LIN {X 0,Y 523.354,Z 614.089,A -85,B 0,C 180,E1 -4766.919,E2 -4766.919} C_VEL
LIN {X 0,Y 523.269,Z 615.476,A -85,B 0,C 180,E1 -4768.459,E2 -4768.459} C_VEL
LIN {X 0,Y 523.242,Z 616,A -85,B 0,C 180,E1 -4769.998,E2 -4769.998} C_VEL
LIN {X 0,Y 523.268,Z 615.478,A -85,B 0,C 180,E1 -4771.537,E2 -4771.537} C_VEL
LIN {X 0,Y 523.353,Z 614.092,A -85,B 0,C 180,E1 -4773.077,E2 -4773.077} C_VEL
LIN {X 0,Y 523.311,Z 611.636,A -85,B 0,C 180,E1 -4774.62,E2 -4774.62} C_VEL
LIN {X 0,Y 523.409,Z 608.259,A -85,B 0,C 180,E1 -4776.164,E2 -4776.164} C_VEL
LIN {X 0,Y 523.505,Z 602.475,A -85,B 0,C 180,E1 -4778.101,E2 -4778.101} C_VEL
LIN {X 0,Y 523.657,Z 594.794,A -85,B 0,C 180,E1 -4780.046,E2 -4780.046} C_VEL
LIN {X 0,Y 523.952,Z 586.574,A -85,B 0,C 180,E1 -4781.713,E2 -4781.713} C_VEL
LIN {X 0,Y 524.219,Z 576.745,A -85,B 0,C 180,E1 -4783.369,E2 -4783.369} C_VEL
LIN {X 0,Y 524.679,Z 566.039,A -85,B 0,C 180,E1 -4784.883,E2 -4784.883} C_VEL
LIN {X 0,Y 525.131,Z 554.075,A -85,B 0,C 180,E1 -4786.32,E2 -4786.32} C_VEL
LIN {X 0,Y 525.732,Z 541.515,A -85,B 0,C 180,E1 -4787.602,E2 -4787.602} C_VEL
LIN {X 0,Y 526.283,Z 529.069,A -85,B 0,C 180,E1 -4788.69,E2 -4788.69} C_VEL
LIN {X 0,Y 526.86,Z 515.69,A -85,B 0,C 180,E1 -4789.68,E2 -4789.68} C_VEL
LIN {X 0,Y 527.439,Z 501.437,A -85,B 0,C 180,E1 -4790.573,E2 -4790.573} C_VEL
LIN {X 0,Y 528.124,Z 485.316,A -85,B 0,C 180,E1 -4791.395,E2 -4791.395} C_VEL
LIN {X 0,Y 528.599,Z 470.295,A -85,B 0,C 180,E1 -4792.007,E2 -4792.007} C_VEL
LIN {X 0,Y 529.013,Z 454.139,A -85,B 0,C 180,E1 -4792.503,E2 -4792.503} C_VEL
LIN {X 0,Y 529.379,Z 437.934,A -85,B 0,C 180,E1 -4792.847,E2 -4792.847} C_VEL
LIN {X 0,Y 530.879,Z 249.022,A -85,B 0,C 180,E1 -4795.545,E2 -4795.545} C_VEL
LIN {X 0,Y 528.181,Z 233.832,A -85,B 0,C 180,E1 -4795.92,E2 -4795.92} C_VEL
LIN {X 0,Y 529.038,Z 210.019,A -85,B 0,C 180,E1 -4798.165,E2 -4798.165} C_VEL
LIN {X 0,Y 523.914,Z 192.537,A -85,B 0,C 180,E1 -4800.198,E2 -4800.198} C_VEL
LIN {X 0,Y 523.925,Z 192.529,A -85,B 0,C 180,E1 -4803.362,E2 -4803.362} C_VEL
LIN {X 0,Y 523.885,Z 192.538,A -85,B 0,C 180,E1 -4806.399,E2 -4806.399} C_VEL
LIN {X 0,Y 523.902,Z 192.542,A -85,B 0,C 180,E1 -4809.082,E2 -4809.082} C_VEL
LIN {X 0,Y 523.931,Z 192.53,A -85,B 0,C 180,E1 -4812.116,E2 -4812.116} C_VEL
LIN {X 0,Y 523.932,Z 192.533,A -85,B 0,C 180,E1 -4815.307,E2 -4815.307} C_VEL
LIN {X 0,Y 523.947,Z 192.531,A -85,B 0,C 180,E1 -4818.686,E2 -4818.686} C_VEL
LIN {X 0,Y 523.894,Z 192.543,A -85,B 0,C 180,E1 -4821.078,E2 -4821.078} C_VEL
LIN {X 0,Y 523.899,Z 192.532,A -85,B 0,C 180,E1 -4823.826,E2 -4823.826} C_VEL
LIN {X 0,Y 523.914,Z 192.536,A -85,B 0,C 180,E1 -4826.634,E2 -4826.634} C_VEL
LIN {X 0,Y 523.926,Z 192.535,A -85,B 0,C 180,E1 -4829.354,E2 -4829.354} C_VEL
LIN {X 0,Y 523.948,Z 192.528,A -85,B 0,C 180,E1 -4832.279,E2 -4832.279} C_VEL
LIN {X 0,Y 523.922,Z 192.528,A -85,B 0,C 180,E1 -4834.58,E2 -4834.58} C_VEL
LIN {X 0,Y 523.921,Z 192.537,A -85,B 0,C 180,E1 -4837.107,E2 -4837.107} C_VEL
LIN {X 0,Y 523.946,Z 192.52,A -85,B 0,C 180,E1 -4839.865,E2 -4839.865} C_VEL
LIN {X 0,Y 523.937,Z 192.535,A -85,B 0,C 180,E1 -4842.837,E2 -4842.837} C_VEL
LIN {X 0,Y 523.942,Z 192.529,A -85,B 0,C 180,E1 -4845.235,E2 -4845.235} C_VEL
LIN {X 0,Y 523.984,Z 192.514,A -85,B 0,C 180,E1 -4848.394,E2 -4848.394} C_VEL
LIN {X 0,Y 523.973,Z 192.525,A -85,B 0,C 180,E1 -4851.516,E2 -4851.516} C_VEL
LIN {X 0,Y 524.066,Z 192.515,A -85,B 0,C 180,E1 -4854.614,E2 -4854.614} C_VEL
LIN {X 0,Y 524.075,Z 192.505,A -85,B 0,C 180,E1 -4857.695,E2 -4857.695} C_VEL
LIN {X 0,Y 524.096,Z 192.517,A -85,B 0,C 180,E1 -4860.769,E2 -4860.769} C_VEL
LIN {X 0,Y 524.044,Z 192.514,A -85,B 0,C 180,E1 -4863.075,E2 -4863.075} C_VEL
LIN {X 0,Y 524.011,Z 192.518,A -85,B 0,C 180,E1 -4866.16,E2 -4866.16} C_VEL
LIN {X 0,Y 523.972,Z 192.524,A -85,B 0,C 180,E1 -4869.263,E2 -4869.263} C_VEL
LIN {X 0,Y 523.975,Z 192.516,A -85,B 0,C 180,E1 -4871.744,E2 -4871.744} C_VEL
LIN {X 0,Y 523.961,Z 192.527,A -85,B 0,C 180,E1 -4875.054,E2 -4875.054} C_VEL
LIN {X 0,Y 523.935,Z 192.527,A -85,B 0,C 180,E1 -4877.97,E2 -4877.97} C_VEL
LIN {X 0,Y 523.943,Z 192.53,A -85,B 0,C 180,E1 -4880.412,E2 -4880.412} C_VEL
LIN {X 0,Y 523.914,Z 192.534,A -85,B 0,C 180,E1 -4882.894,E2 -4882.894} C_VEL
LIN {X 0,Y 523.955,Z 192.524,A -85,B 0,C 180,E1 -4886.022,E2 -4886.022} C_VEL
LIN {X 0,Y 523.913,Z 192.534,A -85,B 0,C 180,E1 -4888.877,E2 -4888.877} C_VEL
LIN {X 0,Y 523.894,Z 192.532,A -85,B 0,C 180,E1 -4891.546,E2 -4891.546} C_VEL
LIN {X 0,Y 523.915,Z 192.535,A -85,B 0,C 180,E1 -4894.292,E2 -4894.292} C_VEL
LIN {X 0,Y 523.887,Z 192.534,A -85,B 0,C 180,E1 -4897.134,E2 -4897.134} C_VEL
LIN {X 0,Y 523.916,Z 192.532,A -85,B 0,C 180,E1 -4900.132,E2 -4900.132} C_VEL
LIN {X 0,Y 523.917,Z 192.537,A -85,B 0,C 180,E1 -4902.462,E2 -4902.462} C_VEL
LIN {X 0,Y 523.924,Z 192.525,A -85,B 0,C 180,E1 -4905.313,E2 -4905.313} C_VEL
LIN {X 0,Y 523.881,Z 192.536,A -85,B 0,C 180,E1 -4906.946,E2 -4906.946} C_VEL
LIN {X 0,Y 523.223,Z 192.62,A -85,B 0,C 180,E1 -4907.588,E2 -4907.588} C_VEL
LIN {X 0,Y 520.388,Z 192.976,A -85,B 0,C 180,E1 -4908.63,E2 -4908.63} C_VEL
LIN {X 0,Y 517.986,Z 193.277,A -85,B 0,C 180,E1 -4909.47,E2 -4909.47} C_VEL
LIN {X 0,Y 516.951,Z 193.403,A -85,B 0,C 180,E1 -4910.118,E2 -4910.118} C_VEL
LIN {X 0,Y 516.864,Z 193.412,A -85,B 0,C 180,E1 -4910.337,E2 -4910.337} C_VEL
LIN {X 0,Y 516.87,Z 193.41,A -85,B 0,C 180,E1 -4913.345,E2 -4913.345} C_VEL
LIN {X 0,Y 516.897,Z 193.41,A -85,B 0,C 180,E1 -4916.124,E2 -4916.124} C_VEL
LIN {X 0,Y 516.88,Z 193.407,A -85,B 0,C 180,E1 -4918.939,E2 -4918.939} C_VEL
LIN {X 0,Y 516.853,Z 193.413,A -85,B 0,C 180,E1 -4921.584,E2 -4921.584} C_VEL
LIN {X 0,Y 516.867,Z 193.414,A -85,B 0,C 180,E1 -4924.211,E2 -4924.211} C_VEL
LIN {X 0,Y 516.851,Z 193.411,A -85,B 0,C 180,E1 -4926.779,E2 -4926.779} C_VEL
LIN {X 0,Y 516.925,Z 193.409,A -85,B 0,C 180,E1 -4929.738,E2 -4929.738} C_VEL
LIN {X 0,Y 516.876,Z 193.411,A -85,B 0,C 180,E1 -4932.597,E2 -4932.597} C_VEL
LIN {X 0,Y 516.934,Z 193.403,A -85,B 0,C 180,E1 -4935.032,E2 -4935.032} C_VEL
LIN {X 0,Y 516.967,Z 193.402,A -85,B 0,C 180,E1 -4938.236,E2 -4938.236} C_VEL
LIN {X 0,Y 516.931,Z 193.406,A -85,B 0,C 180,E1 -4941.401,E2 -4941.401} C_VEL
LIN {X 0,Y 516.986,Z 193.392,A -85,B 0,C 180,E1 -4944.542,E2 -4944.542} C_VEL
LIN {X 0,Y 517.076,Z 193.391,A -85,B 0,C 180,E1 -4947.665,E2 -4947.665} C_VEL
LIN {X 0,Y 516.9,Z 193.516,A -85,B 0,C 180,E1 -4948.979,E2 -4948.979} C_VEL
LIN {X 0,Y 520.755,Z 207.242,A -85,B 0,C 180,E1 -4950.748,E2 -4950.748} C_VEL
LIN {X 0,Y 522.505,Z 211.957,A -85,B 0,C 180,E1 -4950.917,E2 -4950.917} C_VEL
LIN {X 0,Y 524.594,Z 222.487,A -85,B 0,C 180,E1 -4951.189,E2 -4951.189} C_VEL
LIN {X 0,Y 522.849,Z 412.749,A -85,B 0,C 180,E1 -4953.951,E2 -4953.951} C_VEL
LIN {X 0,Y 522.467,Z 429.792,A -85,B 0,C 180,E1 -4954.356,E2 -4954.356} C_VEL
LIN {X 0,Y 521.978,Z 445.68,A -85,B 0,C 180,E1 -4954.892,E2 -4954.892} C_VEL
LIN {X 0,Y 521.408,Z 461.923,A -85,B 0,C 180,E1 -4955.61,E2 -4955.61} C_VEL
LIN {X 0,Y 520.734,Z 477.792,A -85,B 0,C 180,E1 -4956.492,E2 -4956.492} C_VEL
LIN {X 0,Y 520.007,Z 492.311,A -85,B 0,C 180,E1 -4957.476,E2 -4957.476} C_VEL
LIN {X 0,Y 519.365,Z 505.674,A -85,B 0,C 180,E1 -4958.562,E2 -4958.562} C_VEL
LIN {X 0,Y 518.695,Z 518.158,A -85,B 0,C 180,E1 -4959.753,E2 -4959.753} C_VEL
LIN {X 0,Y 518.085,Z 530.572,A -85,B 0,C 180,E1 -4961.147,E2 -4961.147} C_VEL
LIN {X 0,Y 517.568,Z 541.215,A -85,B 0,C 180,E1 -4962.55,E2 -4962.55} C_VEL
LIN {X 0,Y 517.129,Z 551.521,A -85,B 0,C 180,E1 -4964.161,E2 -4964.161} C_VEL
LIN {X 0,Y 516.818,Z 560.197,A -85,B 0,C 180,E1 -4965.783,E2 -4965.783} C_VEL
LIN {X 0,Y 516.551,Z 567.484,A -85,B 0,C 180,E1 -4967.418,E2 -4967.418} C_VEL
LIN {X 0,Y 516.425,Z 573.496,A -85,B 0,C 180,E1 -4969.065,E2 -4969.065} C_VEL
LIN {X 0,Y 516.314,Z 578.28,A -85,B 0,C 180,E1 -4970.728,E2 -4970.728} C_VEL
LIN {X 0,Y 516.194,Z 581.912,A -85,B 0,C 180,E1 -4972.41,E2 -4972.41} C_VEL
LIN {X 0,Y 516.148,Z 584.516,A -85,B 0,C 180,E1 -4974.175,E2 -4974.175} C_VEL
LIN {X 0,Y 516.147,Z 585.934,A -85,B 0,C 180,E1 -4976.015,E2 -4976.015} C_VEL
LIN {X 0,Y 516.178,Z 586.005,A -85,B 0,C 180,E1 -4977.747,E2 -4977.747} C_VEL
LIN {X 0,Y 516.201,Z 585.047,A -85,B 0,C 180,E1 -4979.383,E2 -4979.383} C_VEL
LIN {X 0,Y 516.198,Z 582.857,A -85,B 0,C 180,E1 -4981.157,E2 -4981.157} C_VEL
LIN {X 0,Y 516.284,Z 579.196,A -85,B 0,C 180,E1 -4982.992,E2 -4982.992} C_VEL
LIN {X 0,Y 516.365,Z 574.005,A -85,B 0,C 180,E1 -4984.866,E2 -4984.866} C_VEL
LIN {X 0,Y 516.566,Z 567.745,A -85,B 0,C 180,E1 -4986.61,E2 -4986.61} C_VEL
LIN {X 0,Y 516.818,Z 560.334,A -85,B 0,C 180,E1 -4988.285,E2 -4988.285} C_VEL
LIN {X 0,Y 517.076,Z 552.855,A -85,B 0,C 180,E1 -4989.704,E2 -4989.704} C_VEL
LIN {X 0,Y 517.478,Z 543.552,A -85,B 0,C 180,E1 -4991.201,E2 -4991.201} C_VEL
LIN {X 0,Y 518.049,Z 532.461,A -85,B 0,C 180,E1 -4992.713,E2 -4992.713} C_VEL
LIN {X 0,Y 518.584,Z 520.601,A -85,B 0,C 180,E1 -4994.087,E2 -4994.087} C_VEL
LIN {X 0,Y 519.286,Z 507.484,A -85,B 0,C 180,E1 -4995.374,E2 -4995.374} C_VEL
LIN {X 0,Y 520.013,Z 493.109,A -85,B 0,C 180,E1 -4996.559,E2 -4996.559} C_VEL
LIN {X 0,Y 520.694,Z 478.551,A -85,B 0,C 180,E1 -4997.555,E2 -4997.555} C_VEL
LIN {X 0,Y 521.37,Z 463.096,A -85,B 0,C 180,E1 -4998.425,E2 -4998.425} C_VEL
LIN {X 0,Y 521.918,Z 448.442,A -85,B 0,C 180,E1 -4999.092,E2 -4999.092} C_VEL
LIN {X 0,Y 522.417,Z 432.656,A -85,B 0,C 180,E1 -4999.651,E2 -4999.651} C_VEL
LIN {X 0,Y 522.796,Z 416.77,A -85,B 0,C 180,E1 -5000.056,E2 -5000.056} C_VEL
LIN {X 0,Y 523.05,Z 394.433,A -85,B 0,C 180,E1 -5000.419,E2 -5000.419} C_VEL
LIN {X 0,Y 524.56,Z 221.517,A -85,B 0,C 180,E1 -5002.921,E2 -5002.921} C_VEL
LIN {X 0,Y 522.066,Z 210.261,A -85,B 0,C 180,E1 -5003.227,E2 -5003.227} C_VEL
LIN {X 0,Y 520.905,Z 207.476,A -85,B 0,C 180,E1 -5003.343,E2 -5003.343} C_VEL
LIN {X 0,Y 516.891,Z 193.413,A -85,B 0,C 180,E1 -5005.175,E2 -5005.175} C_VEL
LIN {X 0,Y 516.876,Z 193.415,A -85,B 0,C 180,E1 -5007.975,E2 -5007.975} C_VEL
LIN {X 0,Y 516.923,Z 193.407,A -85,B 0,C 180,E1 -5010.695,E2 -5010.695} C_VEL
LIN {X 0,Y 516.944,Z 193.405,A -85,B 0,C 180,E1 -5013.804,E2 -5013.804} C_VEL
LIN {X 0,Y 516.861,Z 193.414,A -85,B 0,C 180,E1 -5016.776,E2 -5016.776} C_VEL
LIN {X 0,Y 516.939,Z 193.403,A -85,B 0,C 180,E1 -5019.731,E2 -5019.731} C_VEL
LIN {X 0,Y 516.929,Z 193.402,A -85,B 0,C 180,E1 -5022.596,E2 -5022.596} C_VEL
LIN {X 0,Y 516.941,Z 193.401,A -85,B 0,C 180,E1 -5025.03,E2 -5025.03} C_VEL
LIN {X 0,Y 516.965,Z 193.402,A -85,B 0,C 180,E1 -5028.233,E2 -5028.233} C_VEL
LIN {X 0,Y 516.963,Z 193.401,A -85,B 0,C 180,E1 -5031.399,E2 -5031.399} C_VEL
LIN {X 0,Y 517.006,Z 193.399,A -85,B 0,C 180,E1 -5033.756,E2 -5033.756} C_VEL
LIN {X 0,Y 517.079,Z 193.391,A -85,B 0,C 180,E1 -5037.663,E2 -5037.663} C_VEL
LIN {X 0,Y 517.09,Z 193.383,A -85,B 0,C 180,E1 -5040.778,E2 -5040.778} C_VEL
LIN {X 0,Y 517.008,Z 193.394,A -85,B 0,C 180,E1 -5043.117,E2 -5043.117} C_VEL
LIN {X 0,Y 516.999,Z 193.395,A -85,B 0,C 180,E1 -5046.243,E2 -5046.243} C_VEL
LIN {X 0,Y 516.944,Z 193.407,A -85,B 0,C 180,E1 -5049.389,E2 -5049.389} C_VEL
LIN {X 0,Y 516.949,Z 193.404,A -85,B 0,C 180,E1 -5051.807,E2 -5051.807} C_VEL
LIN {X 0,Y 516.941,Z 193.405,A -85,B 0,C 180,E1 -5055.146,E2 -5055.146} C_VEL
LIN {X 0,Y 516.913,Z 193.404,A -85,B 0,C 180,E1 -5058.222,E2 -5058.222} C_VEL
LIN {X 0,Y 516.902,Z 193.407,A -85,B 0,C 180,E1 -5060.702,E2 -5060.702} C_VEL
LIN {X 0,Y 516.887,Z 193.406,A -85,B 0,C 180,E1 -5064.073,E2 -5064.073} C_VEL
LIN {X 0,Y 516.921,Z 193.405,A -85,B 0,C 180,E1 -5066.658,E2 -5066.658} C_VEL
LIN {X 0,Y 516.906,Z 193.41,A -85,B 0,C 180,E1 -5069.523,E2 -5069.523} C_VEL
LIN {X 0,Y 516.892,Z 193.407,A -85,B 0,C 180,E1 -5072.543,E2 -5072.543} C_VEL
LIN {X 0,Y 516.863,Z 193.416,A -85,B 0,C 180,E1 -5075.329,E2 -5075.329} C_VEL
LIN {X 0,Y 516.877,Z 193.409,A -85,B 0,C 180,E1 -5077.942,E2 -5077.942} C_VEL
LIN {X 0,Y 516.881,Z 193.413,A -85,B 0,C 180,E1 -5080.742,E2 -5080.742} C_VEL
LIN {X 0,Y 516.88,Z 193.409,A -85,B 0,C 180,E1 -5083.903,E2 -5083.903} C_VEL
LIN {X 0,Y 516.881,Z 193.411,A -85,B 0,C 180,E1 -5086.107,E2 -5086.107} C_VEL
LIN {X 0,Y 516.861,Z 193.416,A -85,B 0,C 180,E1 -5089.256,E2 -5089.256} C_VEL
LIN {X 0,Y 516.879,Z 193.411,A -85,B 0,C 180,E1 -5092.057,E2 -5092.057} C_VEL
LIN {X 0,Y 516.882,Z 193.415,A -85,B 0,C 180,E1 -5095.174,E2 -5095.174} C_VEL
LIN {X 0,Y 516.872,Z 193.412,A -85,B 0,C 180,E1 -5097.974,E2 -5097.974} C_VEL
LIN {X 0,Y 516.915,Z 193.561,A -85,B 0,C 180,E1 -5099.515,E2 -5099.515} C_VEL
LIN {X 0,Y 522.177,Z 211.476,A -85,B 0,C 180,E1 -5101.622,E2 -5101.622} C_VEL
LIN {X 0,Y 521.632,Z 229.886,A -85,B 0,C 180,E1 -5103.393,E2 -5103.393} C_VEL
LIN {X 0,Y 521.517,Z 233.468,A -85,B 0,C 180,E1 -5103.733,E2 -5103.733} C_VEL
LIN {X 0,Y 524.478,Z 250.611,A -85,B 0,C 180,E1 -5104.151,E2 -5104.151} C_VEL
LIN {X 0,Y 522.764,Z 440.019,A -85,B 0,C 180,E1 -5106.895,E2 -5106.895} C_VEL
LIN {X 0,Y 522.38,Z 456.196,A -85,B 0,C 180,E1 -5107.27,E2 -5107.27} C_VEL
LIN {X 0,Y 521.912,Z 472.323,A -85,B 0,C 180,E1 -5107.796,E2 -5107.796} C_VEL
LIN {X 0,Y 521.414,Z 486.385,A -85,B 0,C 180,E1 -5108.385,E2 -5108.385} C_VEL
LIN {X 0,Y 520.719,Z 500.972,A -85,B 0,C 180,E1 -5109.146,E2 -5109.146} C_VEL
LIN {X 0,Y 520.08,Z 515.268,A -85,B 0,C 180,E1 -5110.048,E2 -5110.048} C_VEL
LIN {X 0,Y 519.445,Z 528.684,A -85,B 0,C 180,E1 -5111.05,E2 -5111.05} C_VEL
LIN {X 0,Y 518.768,Z 542.231,A -85,B 0,C 180,E1 -5112.252,E2 -5112.252} C_VEL
LIN {X 0,Y 518.21,Z 553.745,A -85,B 0,C 180,E1 -5113.452,E2 -5113.452} C_VEL
LIN {X 0,Y 517.67,Z 565.358,A -85,B 0,C 180,E1 -5114.856,E2 -5114.856} C_VEL
LIN {X 0,Y 517.266,Z 575.216,A -85,B 0,C 180,E1 -5116.244,E2 -5116.244} C_VEL
LIN {X 0,Y 516.935,Z 584.745,A -85,B 0,C 180,E1 -5117.833,E2 -5117.833} C_VEL
LIN {X 0,Y 516.674,Z 592.72,A -85,B 0,C 180,E1 -5119.417,E2 -5119.417} C_VEL
LIN {X 0,Y 516.469,Z 599.374,A -85,B 0,C 180,E1 -5120.995,E2 -5120.995} C_VEL
LIN {X 0,Y 516.372,Z 604.769,A -85,B 0,C 180,E1 -5122.569,E2 -5122.569} C_VEL
LIN {X 0,Y 516.321,Z 608.103,A -85,B 0,C 180,E1 -5123.747,E2 -5123.747} C_VEL
LIN {X 0,Y 516.226,Z 611.525,A -85,B 0,C 180,E1 -5125.313,E2 -5125.313} C_VEL
LIN {X 0,Y 516.267,Z 614.015,A -85,B 0,C 180,E1 -5126.877,E2 -5126.877} C_VEL
LIN {X 0,Y 516.186,Z 615.417,A -85,B 0,C 180,E1 -5128.438,E2 -5128.438} C_VEL
LIN {X 0,Y 516.149,Z 615.946,A -85,B 0,C 180,E1 -5129.998,E2 -5129.998} C_VEL
LIN {X 0,Y 516.186,Z 615.419,A -85,B 0,C 180,E1 -5131.558,E2 -5131.558} C_VEL
LIN {X 0,Y 516.266,Z 614.019,A -85,B 0,C 180,E1 -5133.119,E2 -5133.119} C_VEL
LIN {X 0,Y 516.225,Z 611.534,A -85,B 0,C 180,E1 -5134.683,E2 -5134.683} C_VEL
LIN {X 0,Y 516.366,Z 607.42,A -85,B 0,C 180,E1 -5136.505,E2 -5136.505} C_VEL
LIN {X 0,Y 516.42,Z 602.273,A -85,B 0,C 180,E1 -5138.213,E2 -5138.213} C_VEL
LIN {X 0,Y 516.59,Z 594.581,A -85,B 0,C 180,E1 -5140.185,E2 -5140.185} C_VEL
LIN {X 0,Y 516.899,Z 585.9,A -85,B 0,C 180,E1 -5141.964,E2 -5141.964} C_VEL
LIN {X 0,Y 517.199,Z 576.526,A -85,B 0,C 180,E1 -5143.554,E2 -5143.554} C_VEL
LIN {X 0,Y 517.659,Z 566.883,A -85,B 0,C 180,E1 -5144.946,E2 -5144.946} C_VEL
LIN {X 0,Y 518.124,Z 555.641,A -85,B 0,C 180,E1 -5146.345,E2 -5146.345} C_VEL
LIN {X 0,Y 518.773,Z 543.397,A -85,B 0,C 180,E1 -5147.643,E2 -5147.643} C_VEL
LIN {X 0,Y 519.39,Z 530.426,A -85,B 0,C 180,E1 -5148.809,E2 -5148.809} C_VEL
LIN {X 0,Y 520.034,Z 516.878,A -85,B 0,C 180,E1 -5149.847,E2 -5149.847} C_VEL
LIN {X 0,Y 520.634,Z 502.952,A -85,B 0,C 180,E1 -5150.751,E2 -5150.751} C_VEL
LIN {X 0,Y 521.393,Z 487.768,A -85,B 0,C 180,E1 -5151.555,E2 -5151.555} C_VEL
LIN {X 0,Y 521.898,Z 473.922,A -85,B 0,C 180,E1 -5152.148,E2 -5152.148} C_VEL
LIN {X 0,Y 522.354,Z 457.493,A -85,B 0,C 180,E1 -5152.701,E2 -5152.701} C_VEL
LIN {X 0,Y 522.774,Z 441.967,A -85,B 0,C 180,E1 -5153.074,E2 -5153.074} C_VEL
LIN {X 0,Y 523.534,Z 350.102,A -85,B 0,C 180,E1 -5154.42,E2 -5154.42} C_VEL
LIN {X 0,Y 524.462,Z 249.925,A -85,B 0,C 180,E1 -5155.865,E2 -5155.865} C_VEL
LIN {X 0,Y 521.535,Z 233.712,A -85,B 0,C 180,E1 -5156.269,E2 -5156.269} C_VEL
LIN {X 0,Y 522.335,Z 211.716,A -85,B 0,C 180,E1 -5158.374,E2 -5158.374} C_VEL
LIN {X 0,Y 516.899,Z 193.41,A -85,B 0,C 180,E1 -5160.538,E2 -5160.538} C_VEL
LIN {X 0,Y 516.893,Z 193.411,A -85,B 0,C 180,E1 -5163.877,E2 -5163.877} C_VEL
LIN {X 0,Y 516.857,Z 193.416,A -85,B 0,C 180,E1 -5166.744,E2 -5166.744} C_VEL
LIN {X 0,Y 516.862,Z 193.412,A -85,B 0,C 180,E1 -5169.719,E2 -5169.719} C_VEL
LIN {X 0,Y 516.891,Z 193.408,A -85,B 0,C 180,E1 -5171.773,E2 -5171.773} C_VEL
LIN {X 0,Y 516.899,Z 193.412,A -85,B 0,C 180,E1 -5175.008,E2 -5175.008} C_VEL
LIN {X 0,Y 516.898,Z 193.407,A -85,B 0,C 180,E1 -5178.395,E2 -5178.395} C_VEL
LIN {X 0,Y 516.857,Z 193.417,A -85,B 0,C 180,E1 -5181.282,E2 -5181.282} C_VEL
LIN {X 0,Y 516.862,Z 193.408,A -85,B 0,C 180,E1 -5184.219,E2 -5184.219} C_VEL
LIN {X 0,Y 516.868,Z 193.412,A -85,B 0,C 180,E1 -5187.052,E2 -5187.052} C_VEL
LIN {X 0,Y 516.862,Z 193.411,A -85,B 0,C 180,E1 -5189.795,E2 -5189.795} C_VEL
LIN {X 0,Y 516.898,Z 193.408,A -85,B 0,C 180,E1 -5192.466,E2 -5192.466} C_VEL
LIN {X 0,Y 516.881,Z 193.413,A -85,B 0,C 180,E1 -5195.071,E2 -5195.071} C_VEL
LIN {X 0,Y 516.88,Z 193.409,A -85,B 0,C 180,E1 -5197.622,E2 -5197.622} C_VEL
LIN {X 0,Y 516.9,Z 193.398,A -85,B 0,C 180,E1 -5200.129,E2 -5200.129} C_VEL
LIN {X 0,Y 516.897,Z 193.408,A -85,B 0,C 180,E1 -5202.595,E2 -5202.595} C_VEL
LIN {X 0,Y 516.907,Z 193.408,A -85,B 0,C 180,E1 -5205.029,E2 -5205.029} C_VEL
LIN {X 0,Y 516.97,Z 193.385,A -85,B 0,C 180,E1 -5208.234,E2 -5208.234} C_VEL
LIN {X 0,Y 516.938,Z 193.402,A -85,B 0,C 180,E1 -5211.4,E2 -5211.4} C_VEL
LIN {X 0,Y 517.027,Z 193.392,A -85,B 0,C 180,E1 -5214.54,E2 -5214.54} C_VEL
LIN {X 0,Y 517.047,Z 193.38,A -85,B 0,C 180,E1 -5217.663,E2 -5217.663} C_VEL
LIN {X 0,Y 517.065,Z 193.393,A -85,B 0,C 180,E1 -5220.779,E2 -5220.779} C_VEL
LIN {X 0,Y 516.984,Z 193.393,A -85,B 0,C 180,E1 -5223.118,E2 -5223.118} C_VEL
LIN {X 0,Y 516.975,Z 193.395,A -85,B 0,C 180,E1 -5226.244,E2 -5226.244} C_VEL
LIN {X 0,Y 516.926,Z 193.401,A -85,B 0,C 180,E1 -5229.39,E2 -5229.39} C_VEL
LIN {X 0,Y 516.924,Z 193.394,A -85,B 0,C 180,E1 -5231.811,E2 -5231.811} C_VEL
LIN {X 0,Y 516.914,Z 193.404,A -85,B 0,C 180,E1 -5235.149,E2 -5235.149} C_VEL
LIN {X 0,Y 516.896,Z 193.407,A -85,B 0,C 180,E1 -5238.224,E2 -5238.224} C_VEL
LIN {X 0,Y 516.885,Z 193.412,A -85,B 0,C 180,E1 -5240.703,E2 -5240.703} C_VEL
LIN {X 0,Y 516.862,Z 193.41,A -85,B 0,C 180,E1 -5243.224,E2 -5243.224} C_VEL
LIN {X 0,Y 516.914,Z 193.402,A -85,B 0,C 180,E1 -5246.198,E2 -5246.198} C_VEL
LIN {X 0,Y 516.895,Z 193.406,A -85,B 0,C 180,E1 -5249.307,E2 -5249.307} C_VEL
LIN {X 0,Y 516.869,Z 193.409,A -85,B 0,C 180,E1 -5252.546,E2 -5252.546} C_VEL
LIN {X 0,Y 516.855,Z 193.411,A -85,B 0,C 180,E1 -5255.334,E2 -5255.334} C_VEL
LIN {X 0,Y 516.857,Z 193.414,A -85,B 0,C 180,E1 -5257.946,E2 -5257.946} C_VEL
LIN {X 0,Y 516.864,Z 193.412,A -85,B 0,C 180,E1 -5260.744,E2 -5260.744} C_VEL
LIN {X 0,Y 516.863,Z 193.411,A -85,B 0,C 180,E1 -5262.834,E2 -5262.834} C_VEL
LIN {X 0,Y 516.876,Z 193.403,A -85,B 0,C 180,E1 -5265.01,E2 -5265.01} C_VEL
LIN {X 0,Y 516.893,Z 193.411,A -85,B 0,C 180,E1 -5268.402,E2 -5268.402} C_VEL
LIN {X 0,Y 516.864,Z 193.412,A -85,B 0,C 180,E1 -5270.337,E2 -5270.337} C_VEL
LIN {X 0,Y 516.195,Z 193.492,A -85,B 0,C 180,E1 -5270.987,E2 -5270.987} C_VEL
LIN {X 0,Y 513.349,Z 193.852,A -85,B 0,C 180,E1 -5272.043,E2 -5272.043} C_VEL
LIN {X 0,Y 510.942,Z 194.154,A -85,B 0,C 180,E1 -5272.894,E2 -5272.894} C_VEL
LIN {X 0,Y 509.902,Z 194.281,A -85,B 0,C 180,E1 -5273.55,E2 -5273.55} C_VEL
LIN {X 0,Y 509.814,Z 194.29,A -85,B 0,C 180,E1 -5273.773,E2 -5273.773} C_VEL
LIN {X 0,Y 509.848,Z 194.287,A -85,B 0,C 180,E1 -5276.542,E2 -5276.542} C_VEL
LIN {X 0,Y 509.833,Z 194.286,A -85,B 0,C 180,E1 -5279.337,E2 -5279.337} C_VEL
LIN {X 0,Y 509.838,Z 194.294,A -85,B 0,C 180,E1 -5282.055,E2 -5282.055} C_VEL
LIN {X 0,Y 509.797,Z 194.291,A -85,B 0,C 180,E1 -5284.703,E2 -5284.703} C_VEL
LIN {X 0,Y 509.82,Z 194.289,A -85,B 0,C 180,E1 -5287.461,E2 -5287.461} C_VEL
LIN {X 0,Y 509.902,Z 194.286,A -85,B 0,C 180,E1 -5289.847,E2 -5289.847} C_VEL
LIN {X 0,Y 509.85,Z 194.288,A -85,B 0,C 180,E1 -5292.349,E2 -5292.349} C_VEL
LIN {X 0,Y 509.885,Z 194.281,A -85,B 0,C 180,E1 -5294.821,E2 -5294.821} C_VEL
LIN {X 0,Y 509.902,Z 194.282,A -85,B 0,C 180,E1 -5298.127,E2 -5298.127} C_VEL
LIN {X 0,Y 509.885,Z 194.283,A -85,B 0,C 180,E1 -5301.282,E2 -5301.282} C_VEL
LIN {X 0,Y 509.923,Z 194.279,A -85,B 0,C 180,E1 -5303.672,E2 -5303.672} C_VEL
LIN {X 0,Y 509.889,Z 194.283,A -85,B 0,C 180,E1 -5306.842,E2 -5306.842} C_VEL
LIN {X 0,Y 509.925,Z 194.281,A -85,B 0,C 180,E1 -5308.422,E2 -5308.422} C_VEL
LIN {X 0,Y 509.929,Z 194.404,A -85,B 0,C 180,E1 -5308.645,E2 -5308.645} C_VEL
LIN {X 0,Y 513.694,Z 207.744,A -85,B 0,C 180,E1 -5310.366,E2 -5310.366} C_VEL
LIN {X 0,Y 516.341,Z 214.105,A -85,B 0,C 180,E1 -5310.612,E2 -5310.612} C_VEL
LIN {X 0,Y 518.231,Z 223.062,A -85,B 0,C 180,E1 -5310.854,E2 -5310.854} C_VEL
LIN {X 0,Y 516.326,Z 413.678,A -85,B 0,C 180,E1 -5313.66,E2 -5313.66} C_VEL
LIN {X 0,Y 515.912,Z 430.267,A -85,B 0,C 180,E1 -5314.064,E2 -5314.064} C_VEL
LIN {X 0,Y 515.399,Z 445.533,A -85,B 0,C 180,E1 -5314.584,E2 -5314.584} C_VEL
LIN {X 0,Y 514.828,Z 461.086,A -85,B 0,C 180,E1 -5315.272,E2 -5315.272} C_VEL
LIN {X 0,Y 514.177,Z 475.821,A -85,B 0,C 180,E1 -5316.082,E2 -5316.082} C_VEL
LIN {X 0,Y 513.386,Z 490.699,A -85,B 0,C 180,E1 -5317.079,E2 -5317.079} C_VEL
LIN {X 0,Y 512.639,Z 504.363,A -85,B 0,C 180,E1 -5318.179,E2 -5318.179} C_VEL
LIN {X 0,Y 511.923,Z 518.006,A -85,B 0,C 180,E1 -5319.484,E2 -5319.484} C_VEL
LIN {X 0,Y 511.21,Z 530.5,A -85,B 0,C 180,E1 -5320.898,E2 -5320.898} C_VEL
LIN {X 0,Y 510.608,Z 541.859,A -85,B 0,C 180,E1 -5322.418,E2 -5322.418} C_VEL
LIN {X 0,Y 510.158,Z 551.529,A -85,B 0,C 180,E1 -5323.952,E2 -5323.952} C_VEL
LIN {X 0,Y 509.809,Z 560.04,A -85,B 0,C 180,E1 -5325.554,E2 -5325.554} C_VEL
LIN {X 0,Y 509.505,Z 567.558,A -85,B 0,C 180,E1 -5327.253,E2 -5327.253} C_VEL
LIN {X 0,Y 509.368,Z 573.587,A -85,B 0,C 180,E1 -5328.921,E2 -5328.921} C_VEL
LIN {X 0,Y 509.26,Z 578.388,A -85,B 0,C 180,E1 -5330.605,E2 -5330.605} C_VEL
LIN {X 0,Y 509.109,Z 582.113,A -85,B 0,C 180,E1 -5332.345,E2 -5332.345} C_VEL
LIN {X 0,Y 509.047,Z 584.907,A -85,B 0,C 180,E1 -5334.326,E2 -5334.326} C_VEL
LIN {X 0,Y 509.048,Z 586.188,A -85,B 0,C 180,E1 -5336.22,E2 -5336.22} C_VEL
LIN {X 0,Y 509.087,Z 586.164,A -85,B 0,C 180,E1 -5337.995,E2 -5337.995} C_VEL
LIN {X 0,Y 509.098,Z 584.876,A -85,B 0,C 180,E1 -5339.801,E2 -5339.801} C_VEL
LIN {X 0,Y 509.101,Z 582.309,A -85,B 0,C 180,E1 -5341.641,E2 -5341.641} C_VEL
LIN {X 0,Y 509.259,Z 578.346,A -85,B 0,C 180,E1 -5343.506,E2 -5343.506} C_VEL
LIN {X 0,Y 509.377,Z 572.796,A -85,B 0,C 180,E1 -5345.415,E2 -5345.415} C_VEL
LIN {X 0,Y 509.58,Z 566.606,A -85,B 0,C 180,E1 -5347.082,E2 -5347.082} C_VEL
LIN {X 0,Y 509.874,Z 558.569,A -85,B 0,C 180,E1 -5348.842,E2 -5348.842} C_VEL
LIN {X 0,Y 510.243,Z 549.113,A -85,B 0,C 180,E1 -5350.551,E2 -5350.551} C_VEL
LIN {X 0,Y 510.778,Z 538.499,A -85,B 0,C 180,E1 -5352.155,E2 -5352.155} C_VEL
LIN {X 0,Y 511.44,Z 526.579,A -85,B 0,C 180,E1 -5353.671,E2 -5353.671} C_VEL
LIN {X 0,Y 512.106,Z 514.516,A -85,B 0,C 180,E1 -5354.973,E2 -5354.973} C_VEL
LIN {X 0,Y 512.834,Z 501.468,A -85,B 0,C 180,E1 -5356.168,E2 -5356.168} C_VEL
LIN {X 0,Y 513.555,Z 487.161,A -85,B 0,C 180,E1 -5357.271,E2 -5357.271} C_VEL
LIN {X 0,Y 514.285,Z 473.459,A -85,B 0,C 180,E1 -5358.152,E2 -5358.152} C_VEL
LIN {X 0,Y 514.964,Z 457.976,A -85,B 0,C 180,E1 -5358.975,E2 -5358.975} C_VEL
LIN {X 0,Y 515.589,Z 441.818,A -85,B 0,C 180,E1 -5359.651,E2 -5359.651} C_VEL
LIN {X 0,Y 516.076,Z 425.103,A -85,B 0,C 180,E1 -5360.169,E2 -5360.169} C_VEL
LIN {X 0,Y 516.362,Z 409.375,A -85,B 0,C 180,E1 -5360.505,E2 -5360.505} C_VEL
LIN {X 0,Y 518.199,Z 223.799,A -85,B 0,C 180,E1 -5363.232,E2 -5363.232} C_VEL
LIN {X 0,Y 517.241,Z 217.999,A -85,B 0,C 180,E1 -5363.374,E2 -5363.374} C_VEL
LIN {X 0,Y 515.86,Z 212.672,A -85,B 0,C 180,E1 -5363.534,E2 -5363.534} C_VEL
LIN {X 0,Y 513.677,Z 207.591,A -85,B 0,C 180,E1 -5363.757,E2 -5363.757} C_VEL
LIN {X 0,Y 509.866,Z 194.289,A -85,B 0,C 180,E1 -5365.527,E2 -5365.527} C_VEL
LIN {X 0,Y 509.822,Z 194.294,A -85,B 0,C 180,E1 -5368.409,E2 -5368.409} C_VEL
LIN {X 0,Y 509.878,Z 194.282,A -85,B 0,C 180,E1 -5371.155,E2 -5371.155} C_VEL
LIN {X 0,Y 509.91,Z 194.281,A -85,B 0,C 180,E1 -5373.829,E2 -5373.829} C_VEL
LIN {X 0,Y 509.823,Z 194.292,A -85,B 0,C 180,E1 -5376.436,E2 -5376.436} C_VEL
LIN {X 0,Y 509.917,Z 194.279,A -85,B 0,C 180,E1 -5379.844,E2 -5379.844} C_VEL
LIN {X 0,Y 509.883,Z 194.278,A -85,B 0,C 180,E1 -5383.174,E2 -5383.174} C_VEL
LIN {X 0,Y 509.863,Z 194.287,A -85,B 0,C 180,E1 -5385.634,E2 -5385.634} C_VEL
LIN {X 0,Y 509.911,Z 194.277,A -85,B 0,C 180,E1 -5388.874,E2 -5388.874} C_VEL
LIN {X 0,Y 509.949,Z 194.278,A -85,B 0,C 180,E1 -5392.078,E2 -5392.078} C_VEL
LIN {X 0,Y 509.977,Z 194.27,A -85,B 0,C 180,E1 -5394.464,E2 -5394.464} C_VEL
LIN {X 0,Y 510.05,Z 194.266,A -85,B 0,C 180,E1 -5397.63,E2 -5397.63} C_VEL
LIN {X 0,Y 510.051,Z 194.264,A -85,B 0,C 180,E1 -5400,E2 -5400} C_VEL
LIN {X 0,Y 510.048,Z 194.26,A -85,B 0,C 180,E1 -5402.369,E2 -5402.369} C_VEL
LIN {X 0,Y 509.95,Z 194.272,A -85,B 0,C 180,E1 -5406.33,E2 -5406.33} C_VEL
LIN {X 0,Y 509.885,Z 194.286,A -85,B 0,C 180,E1 -5409.52,E2 -5409.52} C_VEL
LIN {X 0,Y 509.902,Z 194.28,A -85,B 0,C 180,E1 -5411.931,E2 -5411.931} C_VEL
LIN {X 0,Y 509.892,Z 194.285,A -85,B 0,C 180,E1 -5415.241,E2 -5415.241} C_VEL
LIN {X 0,Y 509.858,Z 194.283,A -85,B 0,C 180,E1 -5418.483,E2 -5418.483} C_VEL
LIN {X 0,Y 509.843,Z 194.289,A -85,B 0,C 180,E1 -5421.002,E2 -5421.002} C_VEL
LIN {X 0,Y 509.819,Z 194.292,A -85,B 0,C 180,E1 -5423.564,E2 -5423.564} C_VEL
LIN {X 0,Y 509.908,Z 194.277,A -85,B 0,C 180,E1 -5426.378,E2 -5426.378} C_VEL
LIN {X 0,Y 509.87,Z 194.286,A -85,B 0,C 180,E1 -5428.844,E2 -5428.844} C_VEL
LIN {X 0,Y 509.817,Z 194.291,A -85,B 0,C 180,E1 -5431.59,E2 -5431.59} C_VEL
LIN {X 0,Y 509.836,Z 194.286,A -85,B 0,C 180,E1 -5434.414,E2 -5434.414} C_VEL
LIN {X 0,Y 509.814,Z 194.294,A -85,B 0,C 180,E1 -5437.341,E2 -5437.341} C_VEL
LIN {X 0,Y 509.837,Z 194.287,A -85,B 0,C 180,E1 -5440.382,E2 -5440.382} C_VEL
LIN {X 0,Y 509.801,Z 194.299,A -85,B 0,C 180,E1 -5443.059,E2 -5443.059} C_VEL
LIN {X 0,Y 509.822,Z 194.291,A -85,B 0,C 180,E1 -5445.793,E2 -5445.793} C_VEL
LIN {X 0,Y 509.833,Z 194.29,A -85,B 0,C 180,E1 -5448.572,E2 -5448.572} C_VEL
LIN {X 0,Y 509.85,Z 194.286,A -85,B 0,C 180,E1 -5451.786,E2 -5451.786} C_VEL
LIN {X 0,Y 509.828,Z 194.292,A -85,B 0,C 180,E1 -5454.621,E2 -5454.621} C_VEL
LIN {X 0,Y 509.861,Z 194.286,A -85,B 0,C 180,E1 -5457.48,E2 -5457.48} C_VEL
LIN {X 0,Y 509.892,Z 194.466,A -85,B 0,C 180,E1 -5459.162,E2 -5459.162} C_VEL
LIN {X 0,Y 515.605,Z 214.054,A -85,B 0,C 180,E1 -5461.505,E2 -5461.505} C_VEL
LIN {X 0,Y 514.89,Z 233.274,A -85,B 0,C 180,E1 -5463.369,E2 -5463.369} C_VEL
LIN {X 0,Y 518.078,Z 251.318,A -85,B 0,C 180,E1 -5463.821,E2 -5463.821} C_VEL
LIN {X 0,Y 516.209,Z 439.57,A -85,B 0,C 180,E1 -5466.585,E2 -5466.585} C_VEL
LIN {X 0,Y 515.807,Z 455.832,A -85,B 0,C 180,E1 -5466.963,E2 -5466.963} C_VEL
LIN {X 0,Y 515.305,Z 471.998,A -85,B 0,C 180,E1 -5467.496,E2 -5467.496} C_VEL
LIN {X 0,Y 514.748,Z 486.368,A -85,B 0,C 180,E1 -5468.104,E2 -5468.104} C_VEL
LIN {X 0,Y 513.93,Z 502.48,A -85,B 0,C 180,E1 -5468.963,E2 -5468.963} C_VEL
LIN {X 0,Y 513.241,Z 516.427,A -85,B 0,C 180,E1 -5469.875,E2 -5469.875} C_VEL
LIN {X 0,Y 512.512,Z 530.487,A -85,B 0,C 180,E1 -5470.966,E2 -5470.966} C_VEL
LIN {X 0,Y 511.849,Z 543.021,A -85,B 0,C 180,E1 -5472.107,E2 -5472.107} C_VEL
LIN {X 0,Y 511.202,Z 555.293,A -85,B 0,C 180,E1 -5473.424,E2 -5473.424} C_VEL
LIN {X 0,Y 510.657,Z 566.558,A -85,B 0,C 180,E1 -5474.84,E2 -5474.84} C_VEL
LIN {X 0,Y 510.135,Z 577.47,A -85,B 0,C 180,E1 -5476.454,E2 -5476.454} C_VEL
LIN {X 0,Y 509.842,Z 586.644,A -85,B 0,C 180,E1 -5478.065,E2 -5478.065} C_VEL
LIN {X 0,Y 509.537,Z 594.322,A -85,B 0,C 180,E1 -5479.669,E2 -5479.669} C_VEL
LIN {X 0,Y 509.354,Z 602.029,A -85,B 0,C 180,E1 -5481.668,E2 -5481.668} C_VEL
LIN {X 0,Y 509.257,Z 607.889,A -85,B 0,C 180,E1 -5483.66,E2 -5483.66} C_VEL
LIN {X 0,Y 509.142,Z 611.314,A -85,B 0,C 180,E1 -5485.248,E2 -5485.248} C_VEL
LIN {X 0,Y 509.183,Z 613.807,A -85,B 0,C 180,E1 -5486.833,E2 -5486.833} C_VEL
LIN {X 0,Y 509.107,Z 615.211,A -85,B 0,C 180,E1 -5488.416,E2 -5488.416} C_VEL
LIN {X 0,Y 509.061,Z 615.741,A -85,B 0,C 180,E1 -5489.998,E2 -5489.998} C_VEL
LIN {X 0,Y 509.106,Z 615.215,A -85,B 0,C 180,E1 -5491.58,E2 -5491.58} C_VEL
LIN {X 0,Y 509.182,Z 613.815,A -85,B 0,C 180,E1 -5493.163,E2 -5493.163} C_VEL
LIN {X 0,Y 509.141,Z 611.33,A -85,B 0,C 180,E1 -5494.749,E2 -5494.749} C_VEL
LIN {X 0,Y 509.258,Z 607.551,A -85,B 0,C 180,E1 -5496.471,E2 -5496.471} C_VEL
LIN {X 0,Y 509.354,Z 602.065,A -85,B 0,C 180,E1 -5498.328,E2 -5498.328} C_VEL
LIN {X 0,Y 509.534,Z 594.369,A -85,B 0,C 180,E1 -5500.327,E2 -5500.327} C_VEL
LIN {X 0,Y 509.863,Z 585.685,A -85,B 0,C 180,E1 -5502.132,E2 -5502.132} C_VEL
LIN {X 0,Y 510.204,Z 576.308,A -85,B 0,C 180,E1 -5503.743,E2 -5503.743} C_VEL
LIN {X 0,Y 510.682,Z 566.659,A -85,B 0,C 180,E1 -5505.155,E2 -5505.155} C_VEL
LIN {X 0,Y 511.196,Z 555.412,A -85,B 0,C 180,E1 -5506.573,E2 -5506.573} C_VEL
LIN {X 0,Y 511.895,Z 543.165,A -85,B 0,C 180,E1 -5507.888,E2 -5507.888} C_VEL
LIN {X 0,Y 512.606,Z 529.605,A -85,B 0,C 180,E1 -5509.119,E2 -5509.119} C_VEL
LIN {X 0,Y 513.256,Z 516.63,A -85,B 0,C 180,E1 -5510.12,E2 -5510.12} C_VEL
LIN {X 0,Y 513.937,Z 502.694,A -85,B 0,C 180,E1 -5511.034,E2 -5511.034} C_VEL
LIN {X 0,Y 514.78,Z 486.648,A -85,B 0,C 180,E1 -5511.89,E2 -5511.89} C_VEL
LIN {X 0,Y 515.297,Z 472.334,A -85,B 0,C 180,E1 -5512.5,E2 -5512.5} C_VEL
LIN {X 0,Y 515.794,Z 456.259,A -85,B 0,C 180,E1 -5513.033,E2 -5513.033} C_VEL
LIN {X 0,Y 516.254,Z 440.173,A -85,B 0,C 180,E1 -5513.409,E2 -5513.409} C_VEL
LIN {X 0,Y 518.033,Z 250.494,A -85,B 0,C 180,E1 -5516.198,E2 -5516.198} C_VEL
LIN {X 0,Y 514.907,Z 233.414,A -85,B 0,C 180,E1 -5516.643,E2 -5516.643} C_VEL
LIN {X 0,Y 515.734,Z 214.396,A -85,B 0,C 180,E1 -5518.483,E2 -5518.483} C_VEL
LIN {X 0,Y 510.917,Z 197.969,A -85,B 0,C 180,E1 -5520.438,E2 -5520.438} C_VEL
LIN {X 0,Y 509.86,Z 194.288,A -85,B 0,C 180,E1 -5520.912,E2 -5520.912} C_VEL
LIN {X 0,Y 509.844,Z 194.283,A -85,B 0,C 180,E1 -5523.458,E2 -5523.458} C_VEL
LIN {X 0,Y 509.806,Z 194.293,A -85,B 0,C 180,E1 -5526.351,E2 -5526.351} C_VEL
LIN {X 0,Y 509.826,Z 194.292,A -85,B 0,C 180,E1 -5529.35,E2 -5529.35} C_VEL
LIN {X 0,Y 509.811,Z 194.289,A -85,B 0,C 180,E1 -5532.487,E2 -5532.487} C_VEL
LIN {X 0,Y 509.833,Z 194.289,A -85,B 0,C 180,E1 -5535.33,E2 -5535.33} C_VEL
LIN {X 0,Y 509.84,Z 194.288,A -85,B 0,C 180,E1 -5538.573,E2 -5538.573} C_VEL
LIN {X 0,Y 509.825,Z 194.288,A -85,B 0,C 180,E1 -5541.784,E2 -5541.784} C_VEL
LIN {X 0,Y 509.817,Z 194.288,A -85,B 0,C 180,E1 -5544.621,E2 -5544.621} C_VEL
LIN {X 0,Y 509.836,Z 194.281,A -85,B 0,C 180,E1 -5547.479,E2 -5547.479} C_VEL
LIN {X 0,Y 509.828,Z 194.288,A -85,B 0,C 180,E1 -5550.272,E2 -5550.272} C_VEL
LIN {X 0,Y 509.855,Z 194.284,A -85,B 0,C 180,E1 -5552.943,E2 -5552.943} C_VEL
LIN {X 0,Y 509.843,Z 194.286,A -85,B 0,C 180,E1 -5555.573,E2 -5555.573} C_VEL
LIN {X 0,Y 509.822,Z 194.287,A -85,B 0,C 180,E1 -5558.149,E2 -5558.149} C_VEL
LIN {X 0,Y 509.833,Z 194.281,A -85,B 0,C 180,E1 -5560.681,E2 -5560.681} C_VEL
LIN {X 0,Y 509.854,Z 194.288,A -85,B 0,C 180,E1 -5563.174,E2 -5563.174} C_VEL
LIN {X 0,Y 509.83,Z 194.283,A -85,B 0,C 180,E1 -5565.634,E2 -5565.634} C_VEL
LIN {X 0,Y 509.902,Z 194.274,A -85,B 0,C 180,E1 -5568.875,E2 -5568.875} C_VEL
LIN {X 0,Y 509.917,Z 194.276,A -85,B 0,C 180,E1 -5572.078,E2 -5572.078} C_VEL
LIN {X 0,Y 509.974,Z 194.271,A -85,B 0,C 180,E1 -5574.465,E2 -5574.465} C_VEL
LIN {X 0,Y 510.019,Z 194.255,A -85,B 0,C 180,E1 -5577.631,E2 -5577.631} C_VEL
LIN {X 0,Y 510.017,Z 194.263,A -85,B 0,C 180,E1 -5580,E2 -5580} C_VEL
LIN {X 0,Y 510.02,Z 194.267,A -85,B 0,C 180,E1 -5582.37,E2 -5582.37} C_VEL
LIN {X 0,Y 509.943,Z 194.272,A -85,B 0,C 180,E1 -5586.33,E2 -5586.33} C_VEL
LIN {X 0,Y 509.886,Z 194.285,A -85,B 0,C 180,E1 -5588.721,E2 -5588.721} C_VEL
LIN {X 0,Y 509.872,Z 194.273,A -85,B 0,C 180,E1 -5591.933,E2 -5591.933} C_VEL
LIN {X 0,Y 509.861,Z 194.282,A -85,B 0,C 180,E1 -5595.243,E2 -5595.243} C_VEL
LIN {X 0,Y 509.858,Z 194.281,A -85,B 0,C 180,E1 -5598.003,E2 -5598.003} C_VEL
LIN {X 0,Y 509.827,Z 194.288,A -85,B 0,C 180,E1 -5601.003,E2 -5601.003} C_VEL
LIN {X 0,Y 509.821,Z 194.286,A -85,B 0,C 180,E1 -5603.564,E2 -5603.564} C_VEL
LIN {X 0,Y 509.883,Z 194.279,A -85,B 0,C 180,E1 -5606.381,E2 -5606.381} C_VEL
LIN {X 0,Y 509.85,Z 194.287,A -85,B 0,C 180,E1 -5608.846,E2 -5608.846} C_VEL
LIN {X 0,Y 509.793,Z 194.289,A -85,B 0,C 180,E1 -5611.593,E2 -5611.593} C_VEL
LIN {X 0,Y 509.827,Z 194.291,A -85,B 0,C 180,E1 -5614.416,E2 -5614.416} C_VEL
LIN {X 0,Y 509.795,Z 194.29,A -85,B 0,C 180,E1 -5617.343,E2 -5617.343} C_VEL
LIN {X 0,Y 509.817,Z 194.292,A -85,B 0,C 180,E1 -5620.385,E2 -5620.385} C_VEL
LIN {X 0,Y 509.803,Z 194.29,A -85,B 0,C 180,E1 -5623.065,E2 -5623.065} C_VEL
LIN {X 0,Y 509.803,Z 194.286,A -85,B 0,C 180,E1 -5625.796,E2 -5625.796} C_VEL
LIN {X 0,Y 509.836,Z 194.288,A -85,B 0,C 180,E1 -5628.577,E2 -5628.577} C_VEL
LIN {X 0,Y 509.836,Z 194.286,A -85,B 0,C 180,E1 -5631.79,E2 -5631.79} C_VEL
LIN {X 0,Y 509.814,Z 194.29,A -85,B 0,C 180,E1 -5633.773,E2 -5633.773} C_VEL
LIN {X 0,Y 509.15,Z 194.372,A -85,B 0,C 180,E1 -5634.432,E2 -5634.432} C_VEL
LIN {X 0,Y 506.333,Z 194.719,A -85,B 0,C 180,E1 -5635.504,E2 -5635.504} C_VEL
LIN {X 0,Y 503.94,Z 195.025,A -85,B 0,C 180,E1 -5636.368,E2 -5636.368} C_VEL
LIN {X 0,Y 502.891,Z 195.151,A -85,B 0,C 180,E1 -5637.034,E2 -5637.034} C_VEL
LIN {X 0,Y 502.794,Z 195.163,A -85,B 0,C 180,E1 -5637.259,E2 -5637.259} C_VEL
LIN {X 0,Y 502.805,Z 195.164,A -85,B 0,C 180,E1 -5640.068,E2 -5640.068} C_VEL
LIN {X 0,Y 502.804,Z 195.163,A -85,B 0,C 180,E1 -5643.434,E2 -5643.434} C_VEL
LIN {X 0,Y 502.761,Z 195.174,A -85,B 0,C 180,E1 -5646.088,E2 -5646.088} C_VEL
LIN {X 0,Y 502.774,Z 195.167,A -85,B 0,C 180,E1 -5648.691,E2 -5648.691} C_VEL
LIN {X 0,Y 502.804,Z 195.161,A -85,B 0,C 180,E1 -5651.25,E2 -5651.25} C_VEL
LIN {X 0,Y 502.834,Z 195.16,A -85,B 0,C 180,E1 -5654.667,E2 -5654.667} C_VEL
LIN {X 0,Y 502.878,Z 195.158,A -85,B 0,C 180,E1 -5658.042,E2 -5658.042} C_VEL
LIN {X 0,Y 502.85,Z 195.159,A -85,B 0,C 180,E1 -5661.159,E2 -5661.159} C_VEL
LIN {X 0,Y 502.873,Z 195.158,A -85,B 0,C 180,E1 -5663.583,E2 -5663.583} C_VEL
LIN {X 0,Y 502.834,Z 195.162,A -85,B 0,C 180,E1 -5666.797,E2 -5666.797} C_VEL
LIN {X 0,Y 502.915,Z 195.155,A -85,B 0,C 180,E1 -5668.275,E2 -5668.275} C_VEL
LIN {X 0,Y 506.459,Z 207.878,A -85,B 0,C 180,E1 -5669.954,E2 -5669.954} C_VEL
LIN {X 0,Y 510.288,Z 216.803,A -85,B 0,C 180,E1 -5670.314,E2 -5670.314} C_VEL
LIN {X 0,Y 511.866,Z 224.1,A -85,B 0,C 180,E1 -5670.517,E2 -5670.517} C_VEL
LIN {X 0,Y 509.828,Z 413.265,A -85,B 0,C 180,E1 -5673.336,E2 -5673.336} C_VEL
LIN {X 0,Y 509.394,Z 429.682,A -85,B 0,C 180,E1 -5673.735,E2 -5673.735} C_VEL
LIN {X 0,Y 508.889,Z 445.074,A -85,B 0,C 180,E1 -5674.259,E2 -5674.259} C_VEL
LIN {X 0,Y 508.271,Z 460.012,A -85,B 0,C 180,E1 -5674.912,E2 -5674.912} C_VEL
LIN {X 0,Y 507.541,Z 475.463,A -85,B 0,C 180,E1 -5675.763,E2 -5675.763} C_VEL
LIN {X 0,Y 506.687,Z 490.422,A -85,B 0,C 180,E1 -5676.773,E2 -5676.773} C_VEL
LIN {X 0,Y 505.9,Z 504.161,A -85,B 0,C 180,E1 -5677.887,E2 -5677.887} C_VEL
LIN {X 0,Y 505.139,Z 517.492,A -85,B 0,C 180,E1 -5679.168,E2 -5679.168} C_VEL
LIN {X 0,Y 504.438,Z 528.799,A -85,B 0,C 180,E1 -5680.437,E2 -5680.437} C_VEL
LIN {X 0,Y 503.771,Z 539.72,A -85,B 0,C 180,E1 -5681.876,E2 -5681.876} C_VEL
LIN {X 0,Y 503.242,Z 550.325,A -85,B 0,C 180,E1 -5683.529,E2 -5683.529} C_VEL
LIN {X 0,Y 502.912,Z 558.043,A -85,B 0,C 180,E1 -5684.946,E2 -5684.946} C_VEL
LIN {X 0,Y 502.529,Z 565.948,A -85,B 0,C 180,E1 -5686.662,E2 -5686.662} C_VEL
LIN {X 0,Y 502.334,Z 572.12,A -85,B 0,C 180,E1 -5688.307,E2 -5688.307} C_VEL
LIN {X 0,Y 502.275,Z 576.243,A -85,B 0,C 180,E1 -5689.623,E2 -5689.623} C_VEL
LIN {X 0,Y 502.076,Z 580.49,A -85,B 0,C 180,E1 -5691.344,E2 -5691.344} C_VEL
LIN {X 0,Y 501.965,Z 583.626,A -85,B 0,C 180,E1 -5693.082,E2 -5693.082} C_VEL
LIN {X 0,Y 501.964,Z 585.644,A -85,B 0,C 180,E1 -5694.838,E2 -5694.838} C_VEL
LIN {X 0,Y 501.957,Z 586.473,A -85,B 0,C 180,E1 -5696.619,E2 -5696.619} C_VEL
LIN {X 0,Y 501.997,Z 586.165,A -85,B 0,C 180,E1 -5698.426,E2 -5698.426} C_VEL
LIN {X 0,Y 502.035,Z 584.651,A -85,B 0,C 180,E1 -5700.264,E2 -5700.264} C_VEL
LIN {X 0,Y 502.044,Z 581.749,A -85,B 0,C 180,E1 -5702.138,E2 -5702.138} C_VEL
LIN {X 0,Y 502.188,Z 577.407,A -85,B 0,C 180,E1 -5704.042,E2 -5704.042} C_VEL
LIN {X 0,Y 502.34,Z 572.224,A -85,B 0,C 180,E1 -5705.761,E2 -5705.761} C_VEL
LIN {X 0,Y 502.587,Z 565.591,A -85,B 0,C 180,E1 -5707.52,E2 -5707.52} C_VEL
LIN {X 0,Y 502.911,Z 557.951,A -85,B 0,C 180,E1 -5709.174,E2 -5709.174} C_VEL
LIN {X 0,Y 503.264,Z 549.211,A -85,B 0,C 180,E1 -5710.758,E2 -5710.758} C_VEL
LIN {X 0,Y 503.839,Z 538.97,A -85,B 0,C 180,E1 -5712.328,E2 -5712.328} C_VEL
LIN {X 0,Y 504.534,Z 527.589,A -85,B 0,C 180,E1 -5713.807,E2 -5713.807} C_VEL
LIN {X 0,Y 505.273,Z 515.093,A -85,B 0,C 180,E1 -5715.185,E2 -5715.185} C_VEL
LIN {X 0,Y 506.04,Z 502.242,A -85,B 0,C 180,E1 -5716.38,E2 -5716.38} C_VEL
LIN {X 0,Y 506.796,Z 488.653,A -85,B 0,C 180,E1 -5717.452,E2 -5717.452} C_VEL
LIN {X 0,Y 507.608,Z 474.523,A -85,B 0,C 180,E1 -5718.387,E2 -5718.387} C_VEL
LIN {X 0,Y 508.306,Z 459.688,A -85,B 0,C 180,E1 -5719.2,E2 -5719.2} C_VEL
LIN {X 0,Y 508.957,Z 443.619,A -85,B 0,C 180,E1 -5719.893,E2 -5719.893} C_VEL
LIN {X 0,Y 509.445,Z 427.753,A -85,B 0,C 180,E1 -5720.412,E2 -5720.412} C_VEL
LIN {X 0,Y 509.859,Z 410.333,A -85,B 0,C 180,E1 -5720.806,E2 -5720.806} C_VEL
LIN {X 0,Y 511.862,Z 224.834,A -85,B 0,C 180,E1 -5723.57,E2 -5723.57} C_VEL
LIN {X 0,Y 509.976,Z 215.661,A -85,B 0,C 180,E1 -5723.822,E2 -5723.822} C_VEL
LIN {X 0,Y 506.477,Z 207.878,A -85,B 0,C 180,E1 -5724.168,E2 -5724.168} C_VEL
LIN {X 0,Y 502.82,Z 195.168,A -85,B 0,C 180,E1 -5725.911,E2 -5725.911} C_VEL
LIN {X 0,Y 502.798,Z 195.167,A -85,B 0,C 180,E1 -5728.856,E2 -5728.856} C_VEL
LIN {X 0,Y 502.846,Z 195.159,A -85,B 0,C 180,E1 -5731.704,E2 -5731.704} C_VEL
LIN {X 0,Y 502.823,Z 195.167,A -85,B 0,C 180,E1 -5734.323,E2 -5734.323} C_VEL
LIN {X 0,Y 502.804,Z 195.165,A -85,B 0,C 180,E1 -5737.297,E2 -5737.297} C_VEL
LIN {X 0,Y 502.826,Z 195.165,A -85,B 0,C 180,E1 -5740.4,E2 -5740.4} C_VEL
LIN {X 0,Y 502.833,Z 195.156,A -85,B 0,C 180,E1 -5742.931,E2 -5742.931} C_VEL
LIN {X 0,Y 502.844,Z 195.159,A -85,B 0,C 180,E1 -5745.429,E2 -5745.429} C_VEL
LIN {X 0,Y 502.875,Z 195.154,A -85,B 0,C 180,E1 -5748.716,E2 -5748.716} C_VEL
LIN {X 0,Y 502.899,Z 195.157,A -85,B 0,C 180,E1 -5751.966,E2 -5751.966} C_VEL
LIN {X 0,Y 502.934,Z 195.148,A -85,B 0,C 180,E1 -5754.386,E2 -5754.386} C_VEL
LIN {X 0,Y 503.02,Z 195.141,A -85,B 0,C 180,E1 -5757.597,E2 -5757.597} C_VEL
LIN {X 0,Y 503.023,Z 195.14,A -85,B 0,C 180,E1 -5760,E2 -5760} C_VEL
LIN {X 0,Y 503.019,Z 195.136,A -85,B 0,C 180,E1 -5762.402,E2 -5762.402} C_VEL
LIN {X 0,Y 502.928,Z 195.153,A -85,B 0,C 180,E1 -5765.613,E2 -5765.613} C_VEL
LIN {X 0,Y 502.878,Z 195.156,A -85,B 0,C 180,E1 -5768.033,E2 -5768.033} C_VEL
LIN {X 0,Y 502.874,Z 195.157,A -85,B 0,C 180,E1 -5771.283,E2 -5771.283} C_VEL
LIN {X 0,Y 502.841,Z 195.158,A -85,B 0,C 180,E1 -5774.571,E2 -5774.571} C_VEL
LIN {X 0,Y 502.819,Z 195.162,A -85,B 0,C 180,E1 -5777.908,E2 -5777.908} C_VEL
LIN {X 0,Y 502.827,Z 195.16,A -85,B 0,C 180,E1 -5780.536,E2 -5780.536} C_VEL
LIN {X 0,Y 502.786,Z 195.168,A -85,B 0,C 180,E1 -5783.04,E2 -5783.04} C_VEL
LIN {X 0,Y 502.818,Z 195.164,A -85,B 0,C 180,E1 -5785.676,E2 -5785.676} C_VEL
LIN {X 0,Y 502.835,Z 195.159,A -85,B 0,C 180,E1 -5788.373,E2 -5788.373} C_VEL
LIN {X 0,Y 502.79,Z 195.167,A -85,B 0,C 180,E1 -5791.498,E2 -5791.498} C_VEL
LIN {X 0,Y 502.789,Z 195.164,A -85,B 0,C 180,E1 -5794.441,E2 -5794.441} C_VEL
LIN {X 0,Y 502.776,Z 195.173,A -85,B 0,C 180,E1 -5797.177,E2 -5797.177} C_VEL
LIN {X 0,Y 502.786,Z 195.165,A -85,B 0,C 180,E1 -5800.015,E2 -5800.015} C_VEL
LIN {X 0,Y 502.803,Z 195.162,A -85,B 0,C 180,E1 -5802.199,E2 -5802.199} C_VEL
LIN {X 0,Y 502.785,Z 195.17,A -85,B 0,C 180,E1 -5805.47,E2 -5805.47} C_VEL
LIN {X 0,Y 502.795,Z 195.163,A -85,B 0,C 180,E1 -5807.86,E2 -5807.86} C_VEL
LIN {X 0,Y 502.797,Z 195.17,A -85,B 0,C 180,E1 -5811.023,E2 -5811.023} C_VEL
LIN {X 0,Y 502.772,Z 195.17,A -85,B 0,C 180,E1 -5814.169,E2 -5814.169} C_VEL
LIN {X 0,Y 502.834,Z 195.166,A -85,B 0,C 180,E1 -5816.993,E2 -5816.993} C_VEL
LIN {X 0,Y 502.842,Z 195.357,A -85,B 0,C 180,E1 -5818.793,E2 -5818.793} C_VEL
LIN {X 0,Y 508.34,Z 213.844,A -85,B 0,C 180,E1 -5821.059,E2 -5821.059} C_VEL
LIN {X 0,Y 508.998,Z 217.185,A -85,B 0,C 180,E1 -5821.439,E2 -5821.439} C_VEL
LIN {X 0,Y 508.262,Z 232.914,A -85,B 0,C 180,E1 -5822.981,E2 -5822.981} C_VEL
LIN {X 0,Y 511.705,Z 253.143,A -85,B 0,C 180,E1 -5823.5,E2 -5823.5} C_VEL
LIN {X 0,Y 509.672,Z 440.645,A -85,B 0,C 180,E1 -5826.293,E2 -5826.293} C_VEL
LIN {X 0,Y 509.221,Z 457.314,A -85,B 0,C 180,E1 -5826.702,E2 -5826.702} C_VEL
LIN {X 0,Y 508.643,Z 472.983,A -85,B 0,C 180,E1 -5827.238,E2 -5827.238} C_VEL
LIN {X 0,Y 508.068,Z 487.097,A -85,B 0,C 180,E1 -5827.855,E2 -5827.855} C_VEL
LIN {X 0,Y 507.224,Z 502.429,A -85,B 0,C 180,E1 -5828.686,E2 -5828.686} C_VEL
LIN {X 0,Y 506.492,Z 516.15,A -85,B 0,C 180,E1 -5829.595,E2 -5829.595} C_VEL
LIN {X 0,Y 505.669,Z 530.678,A -85,B 0,C 180,E1 -5830.739,E2 -5830.739} C_VEL
LIN {X 0,Y 504.933,Z 543.749,A -85,B 0,C 180,E1 -5831.958,E2 -5831.958} C_VEL
LIN {X 0,Y 504.276,Z 555.041,A -85,B 0,C 180,E1 -5833.189,E2 -5833.189} C_VEL
LIN {X 0,Y 503.68,Z 566.315,A -85,B 0,C 180,E1 -5834.625,E2 -5834.625} C_VEL
LIN {X 0,Y 503.15,Z 577.234,A -85,B 0,C 180,E1 -5836.262,E2 -5836.262} C_VEL
LIN {X 0,Y 502.791,Z 586.414,A -85,B 0,C 180,E1 -5837.896,E2 -5837.896} C_VEL
LIN {X 0,Y 502.485,Z 594.097,A -85,B 0,C 180,E1 -5839.522,E2 -5839.522} C_VEL
LIN {X 0,Y 502.258,Z 601.809,A -85,B 0,C 180,E1 -5841.55,E2 -5841.55} C_VEL
LIN {X 0,Y 502.184,Z 607.675,A -85,B 0,C 180,E1 -5843.57,E2 -5843.57} C_VEL
LIN {X 0,Y 502.062,Z 611.103,A -85,B 0,C 180,E1 -5845.18,E2 -5845.18} C_VEL
LIN {X 0,Y 502.101,Z 613.6,A -85,B 0,C 180,E1 -5846.789,E2 -5846.789} C_VEL
LIN {X 0,Y 502.031,Z 615.005,A -85,B 0,C 180,E1 -5848.394,E2 -5848.394} C_VEL
LIN {X 0,Y 501.975,Z 615.537,A -85,B 0,C 180,E1 -5849.998,E2 -5849.998} C_VEL
LIN {X 0,Y 502.03,Z 615.011,A -85,B 0,C 180,E1 -5851.602,E2 -5851.602} C_VEL
LIN {X 0,Y 502.1,Z 613.611,A -85,B 0,C 180,E1 -5853.208,E2 -5853.208} C_VEL
LIN {X 0,Y 502.06,Z 611.125,A -85,B 0,C 180,E1 -5854.816,E2 -5854.816} C_VEL
LIN {X 0,Y 502.18,Z 607.6,A -85,B 0,C 180,E1 -5856.467,E2 -5856.467} C_VEL
LIN {X 0,Y 502.259,Z 601.856,A -85,B 0,C 180,E1 -5858.446,E2 -5858.446} C_VEL
LIN {X 0,Y 502.487,Z 594.157,A -85,B 0,C 180,E1 -5860.474,E2 -5860.474} C_VEL
LIN {X 0,Y 502.834,Z 585.47,A -85,B 0,C 180,E1 -5862.304,E2 -5862.304} C_VEL
LIN {X 0,Y 503.199,Z 576.089,A -85,B 0,C 180,E1 -5863.939,E2 -5863.939} C_VEL
LIN {X 0,Y 503.713,Z 566.436,A -85,B 0,C 180,E1 -5865.37,E2 -5865.37} C_VEL
LIN {X 0,Y 504.273,Z 555.183,A -85,B 0,C 180,E1 -5866.807,E2 -5866.807} C_VEL
LIN {X 0,Y 505.012,Z 542.932,A -85,B 0,C 180,E1 -5868.14,E2 -5868.14} C_VEL
LIN {X 0,Y 505.77,Z 529.602,A -85,B 0,C 180,E1 -5869.367,E2 -5869.367} C_VEL
LIN {X 0,Y 506.511,Z 516.383,A -85,B 0,C 180,E1 -5870.4,E2 -5870.4} C_VEL
LIN {X 0,Y 507.237,Z 502.645,A -85,B 0,C 180,E1 -5871.312,E2 -5871.312} C_VEL
LIN {X 0,Y 508.067,Z 487.796,A -85,B 0,C 180,E1 -5872.12,E2 -5872.12} C_VEL
LIN {X 0,Y 508.65,Z 473.353,A -85,B 0,C 180,E1 -5872.757,E2 -5872.757} C_VEL
LIN {X 0,Y 509.226,Z 456.861,A -85,B 0,C 180,E1 -5873.321,E2 -5873.321} C_VEL
LIN {X 0,Y 509.712,Z 441.252,A -85,B 0,C 180,E1 -5873.701,E2 -5873.701} C_VEL
LIN {X 0,Y 511.611,Z 262.47,A -85,B 0,C 180,E1 -5876.362,E2 -5876.362} C_VEL
LIN {X 0,Y 511.587,Z 251.388,A -85,B 0,C 180,E1 -5876.536,E2 -5876.536} C_VEL
LIN {X 0,Y 508.315,Z 233.3,A -85,B 0,C 180,E1 -5877.007,E2 -5877.007} C_VEL
LIN {X 0,Y 509.092,Z 216.423,A -85,B 0,C 180,E1 -5878.664,E2 -5878.664} C_VEL
LIN {X 0,Y 503.917,Z 198.818,A -85,B 0,C 180,E1 -5880.794,E2 -5880.794} C_VEL
LIN {X 0,Y 502.801,Z 195.17,A -85,B 0,C 180,E1 -5881.272,E2 -5881.272} C_VEL
LIN {X 0,Y 502.789,Z 195.168,A -85,B 0,C 180,E1 -5883.991,E2 -5883.991} C_VEL
LIN {X 0,Y 502.758,Z 195.173,A -85,B 0,C 180,E1 -5887.175,E2 -5887.175} C_VEL
LIN {X 0,Y 502.767,Z 195.166,A -85,B 0,C 180,E1 -5890.013,E2 -5890.013} C_VEL
LIN {X 0,Y 502.781,Z 195.164,A -85,B 0,C 180,E1 -5892.197,E2 -5892.197} C_VEL
LIN {X 0,Y 502.777,Z 195.166,A -85,B 0,C 180,E1 -5895.466,E2 -5895.466} C_VEL
LIN {X 0,Y 502.805,Z 195.163,A -85,B 0,C 180,E1 -5897.862,E2 -5897.862} C_VEL
LIN {X 0,Y 502.776,Z 195.172,A -85,B 0,C 180,E1 -5901.022,E2 -5901.022} C_VEL
LIN {X 0,Y 502.757,Z 195.165,A -85,B 0,C 180,E1 -5904.166,E2 -5904.166} C_VEL
LIN {X 0,Y 502.804,Z 195.164,A -85,B 0,C 180,E1 -5906.991,E2 -5906.991} C_VEL
LIN {X 0,Y 502.785,Z 195.165,A -85,B 0,C 180,E1 -5910.063,E2 -5910.063} C_VEL
LIN {X 0,Y 502.803,Z 195.164,A -85,B 0,C 180,E1 -5912.532,E2 -5912.532} C_VEL
LIN {X 0,Y 502.799,Z 195.166,A -85,B 0,C 180,E1 -5915.297,E2 -5915.297} C_VEL
LIN {X 0,Y 502.789,Z 195.163,A -85,B 0,C 180,E1 -5917.827,E2 -5917.827} C_VEL
LIN {X 0,Y 502.793,Z 195.156,A -85,B 0,C 180,E1 -5920.399,E2 -5920.399} C_VEL
LIN {X 0,Y 502.803,Z 195.169,A -85,B 0,C 180,E1 -5922.931,E2 -5922.931} C_VEL
LIN {X 0,Y 502.811,Z 195.159,A -85,B 0,C 180,E1 -5925.429,E2 -5925.429} C_VEL
LIN {X 0,Y 502.868,Z 195.146,A -85,B 0,C 180,E1 -5928.717,E2 -5928.717} C_VEL
LIN {X 0,Y 502.868,Z 195.154,A -85,B 0,C 180,E1 -5931.967,E2 -5931.967} C_VEL
LIN {X 0,Y 502.926,Z 195.147,A -85,B 0,C 180,E1 -5934.387,E2 -5934.387} C_VEL
LIN {X 0,Y 502.989,Z 195.13,A -85,B 0,C 180,E1 -5937.598,E2 -5937.598} C_VEL
LIN {X 0,Y 502.989,Z 195.138,A -85,B 0,C 180,E1 -5940,E2 -5940} C_VEL
LIN {X 0,Y 502.99,Z 195.143,A -85,B 0,C 180,E1 -5942.403,E2 -5942.403} C_VEL
LIN {X 0,Y 502.914,Z 195.143,A -85,B 0,C 180,E1 -5945.614,E2 -5945.614} C_VEL
LIN {X 0,Y 502.869,Z 195.155,A -85,B 0,C 180,E1 -5948.034,E2 -5948.034} C_VEL
LIN {X 0,Y 502.849,Z 195.147,A -85,B 0,C 180,E1 -5951.284,E2 -5951.284} C_VEL
LIN {X 0,Y 502.819,Z 195.166,A -85,B 0,C 180,E1 -5954.572,E2 -5954.572} C_VEL
LIN {X 0,Y 502.832,Z 195.155,A -85,B 0,C 180,E1 -5957.909,E2 -5957.909} C_VEL
LIN {X 0,Y 502.8,Z 195.165,A -85,B 0,C 180,E1 -5960.539,E2 -5960.539} C_VEL
LIN {X 0,Y 502.777,Z 195.165,A -85,B 0,C 180,E1 -5963.042,E2 -5963.042} C_VEL
LIN {X 0,Y 502.812,Z 195.154,A -85,B 0,C 180,E1 -5965.678,E2 -5965.678} C_VEL
LIN {X 0,Y 502.813,Z 195.166,A -85,B 0,C 180,E1 -5968.375,E2 -5968.375} C_VEL
LIN {X 0,Y 502.766,Z 195.164,A -85,B 0,C 180,E1 -5971.501,E2 -5971.501} C_VEL
LIN {X 0,Y 502.781,Z 195.162,A -85,B 0,C 180,E1 -5973.996,E2 -5973.996} C_VEL
LIN {X 0,Y 502.757,Z 195.167,A -85,B 0,C 180,E1 -5977.181,E2 -5977.181} C_VEL
LIN {X 0,Y 502.765,Z 195.163,A -85,B 0,C 180,E1 -5980.018,E2 -5980.018} C_VEL
LIN {X 0,Y 502.783,Z 195.172,A -85,B 0,C 180,E1 -5982.202,E2 -5982.202} C_VEL
LIN {X 0,Y 502.767,Z 195.16,A -85,B 0,C 180,E1 -5985.473,E2 -5985.473} C_VEL
LIN {X 0,Y 502.778,Z 195.169,A -85,B 0,C 180,E1 -5987.863,E2 -5987.863} C_VEL
LIN {X 0,Y 502.786,Z 195.16,A -85,B 0,C 180,E1 -5991.027,E2 -5991.027} C_VEL
LIN {X 0,Y 502.769,Z 195.17,A -85,B 0,C 180,E1 -5994.171,E2 -5994.171} C_VEL
LIN {X 0,Y 502.794,Z 195.163,A -85,B 0,C 180,E1 -5997.259,E2 -5997.259} C_VEL
LIN {X 0,Y 502.096,Z 195.256,A -85,B 0,C 180,E1 -5997.928,E2 -5997.928} C_VEL
LIN {X 0,Y 499.233,Z 195.609,A -85,B 0,C 180,E1 -5999.014,E2 -5999.014} C_VEL
LIN {X 0,Y 496.835,Z 195.908,A -85,B 0,C 180,E1 -5999.889,E2 -5999.889} C_VEL
LIN {X 0,Y 495.809,Z 196.034,A -85,B 0,C 180,E1 -6000.565,E2 -6000.565} C_VEL
LIN {X 0,Y 495.727,Z 196.042,A -85,B 0,C 180,E1 -6000.793,E2 -6000.793} C_VEL
LIN {X 0,Y 495.724,Z 196.047,A -85,B 0,C 180,E1 -6003.932,E2 -6003.932} C_VEL
LIN {X 0,Y 495.753,Z 196.039,A -85,B 0,C 180,E1 -6007.143,E2 -6007.143} C_VEL
LIN {X 0,Y 495.756,Z 196.044,A -85,B 0,C 180,E1 -6010.112,E2 -6010.112} C_VEL
LIN {X 0,Y 495.711,Z 196.047,A -85,B 0,C 180,E1 -6012.681,E2 -6012.681} C_VEL
LIN {X 0,Y 495.778,Z 196.04,A -85,B 0,C 180,E1 -6015.219,E2 -6015.219} C_VEL
LIN {X 0,Y 495.851,Z 196.03,A -85,B 0,C 180,E1 -6018.557,E2 -6018.557} C_VEL
LIN {X 0,Y 495.815,Z 196.038,A -85,B 0,C 180,E1 -6021.853,E2 -6021.853} C_VEL
LIN {X 0,Y 495.857,Z 196.023,A -85,B 0,C 180,E1 -6024.308,E2 -6024.308} C_VEL
LIN {X 0,Y 495.9,Z 196.028,A -85,B 0,C 180,E1 -6027.921,E2 -6027.921} C_VEL
LIN {X 0,Y 499.38,Z 208.197,A -85,B 0,C 180,E1 -6029.542,E2 -6029.542} C_VEL
LIN {X 0,Y 504.295,Z 219.491,A -85,B 0,C 180,E1 -6030.013,E2 -6030.013} C_VEL
LIN {X 0,Y 505.492,Z 225.443,A -85,B 0,C 180,E1 -6030.176,E2 -6030.176} C_VEL
LIN {X 0,Y 503.332,Z 414.159,A -85,B 0,C 180,E1 -6033.028,E2 -6033.028} C_VEL
LIN {X 0,Y 502.847,Z 431.21,A -85,B 0,C 180,E1 -6033.457,E2 -6033.457} C_VEL
LIN {X 0,Y 502.224,Z 446.94,A -85,B 0,C 180,E1 -6034.014,E2 -6034.014} C_VEL
LIN {X 0,Y 501.57,Z 462.365,A -85,B 0,C 180,E1 -6034.724,E2 -6034.724} C_VEL
LIN {X 0,Y 500.81,Z 476.981,A -85,B 0,C 180,E1 -6035.553,E2 -6035.553} C_VEL
LIN {X 0,Y 499.94,Z 491.529,A -85,B 0,C 180,E1 -6036.56,E2 -6036.56} C_VEL
LIN {X 0,Y 499.082,Z 505.129,A -85,B 0,C 180,E1 -6037.69,E2 -6037.69} C_VEL
LIN {X 0,Y 498.305,Z 517.759,A -85,B 0,C 180,E1 -6038.927,E2 -6038.927} C_VEL
LIN {X 0,Y 497.575,Z 528.731,A -85,B 0,C 180,E1 -6040.171,E2 -6040.171} C_VEL
LIN {X 0,Y 496.878,Z 539.681,A -85,B 0,C 180,E1 -6041.63,E2 -6041.63} C_VEL
LIN {X 0,Y 496.339,Z 549.084,A -85,B 0,C 180,E1 -6043.096,E2 -6043.096} C_VEL
LIN {X 0,Y 495.908,Z 558.265,A -85,B 0,C 180,E1 -6044.781,E2 -6044.781} C_VEL
LIN {X 0,Y 495.512,Z 566.003,A -85,B 0,C 180,E1 -6046.481,E2 -6046.481} C_VEL
LIN {X 0,Y 495.286,Z 572.35,A -85,B 0,C 180,E1 -6048.192,E2 -6048.192} C_VEL
LIN {X 0,Y 495.169,Z 577.498,A -85,B 0,C 180,E1 -6049.917,E2 -6049.917} C_VEL
LIN {X 0,Y 494.955,Z 581.549,A -85,B 0,C 180,E1 -6051.666,E2 -6051.666} C_VEL
LIN {X 0,Y 494.856,Z 584.381,A -85,B 0,C 180,E1 -6053.433,E2 -6053.433} C_VEL
LIN {X 0,Y 494.856,Z 586.119,A -85,B 0,C 180,E1 -6055.219,E2 -6055.219} C_VEL
LIN {X 0,Y 494.875,Z 586.754,A -85,B 0,C 180,E1 -6057.031,E2 -6057.031} C_VEL
LIN {X 0,Y 494.909,Z 586.126,A -85,B 0,C 180,E1 -6058.871,E2 -6058.871} C_VEL
LIN {X 0,Y 494.94,Z 584.278,A -85,B 0,C 180,E1 -6060.744,E2 -6060.744} C_VEL
LIN {X 0,Y 494.993,Z 581.088,A -85,B 0,C 180,E1 -6062.653,E2 -6062.653} C_VEL
LIN {X 0,Y 495.121,Z 577.721,A -85,B 0,C 180,E1 -6064.099,E2 -6064.099} C_VEL
LIN {X 0,Y 495.301,Z 571.971,A -85,B 0,C 180,E1 -6066.021,E2 -6066.021} C_VEL
LIN {X 0,Y 495.586,Z 565.105,A -85,B 0,C 180,E1 -6067.832,E2 -6067.832} C_VEL
LIN {X 0,Y 496,Z 556.8,A -85,B 0,C 180,E1 -6069.615,E2 -6069.615} C_VEL
LIN {X 0,Y 496.502,Z 546.8,A -85,B 0,C 180,E1 -6071.39,E2 -6071.39} C_VEL
LIN {X 0,Y 497.182,Z 535.882,A -85,B 0,C 180,E1 -6073.004,E2 -6073.004} C_VEL
LIN {X 0,Y 497.87,Z 524.046,A -85,B 0,C 180,E1 -6074.483,E2 -6074.483} C_VEL
LIN {X 0,Y 498.719,Z 511.315,A -85,B 0,C 180,E1 -6075.83,E2 -6075.83} C_VEL
LIN {X 0,Y 499.582,Z 498.11,A -85,B 0,C 180,E1 -6077.015,E2 -6077.015} C_VEL
LIN {X 0,Y 500.46,Z 483.768,A -85,B 0,C 180,E1 -6078.098,E2 -6078.098} C_VEL
LIN {X 0,Y 501.311,Z 468.688,A -85,B 0,C 180,E1 -6079.037,E2 -6079.037} C_VEL
LIN {X 0,Y 502.01,Z 453.475,A -85,B 0,C 180,E1 -6079.802,E2 -6079.802} C_VEL
LIN {X 0,Y 502.651,Z 436.935,A -85,B 0,C 180,E1 -6080.451,E2 -6080.451} C_VEL
LIN {X 0,Y 503.192,Z 420.524,A -85,B 0,C 180,E1 -6080.921,E2 -6080.921} C_VEL
LIN {X 0,Y 503.489,Z 402.916,A -85,B 0,C 180,E1 -6081.255,E2 -6081.255} C_VEL
LIN {X 0,Y 505.489,Z 224.925,A -85,B 0,C 180,E1 -6083.936,E2 -6083.936} C_VEL
LIN {X 0,Y 503.78,Z 217.939,A -85,B 0,C 180,E1 -6084.148,E2 -6084.148} C_VEL
LIN {X 0,Y 499.305,Z 208.196,A -85,B 0,C 180,E1 -6084.586,E2 -6084.586} C_VEL
LIN {X 0,Y 495.78,Z 196.042,A -85,B 0,C 180,E1 -6086.284,E2 -6086.284} C_VEL
LIN {X 0,Y 495.754,Z 196.044,A -85,B 0,C 180,E1 -6089.312,E2 -6089.312} C_VEL
LIN {X 0,Y 495.783,Z 196.041,A -85,B 0,C 180,E1 -6092.108,E2 -6092.108} C_VEL
LIN {X 0,Y 495.754,Z 196.045,A -85,B 0,C 180,E1 -6094.83,E2 -6094.83} C_VEL
LIN {X 0,Y 495.749,Z 196.045,A -85,B 0,C 180,E1 -6097.494,E2 -6097.494} C_VEL
LIN {X 0,Y 495.772,Z 196.044,A -85,B 0,C 180,E1 -6100.109,E2 -6100.109} C_VEL
LIN {X 0,Y 495.786,Z 196.034,A -85,B 0,C 180,E1 -6102.681,E2 -6102.681} C_VEL
LIN {X 0,Y 495.789,Z 196.037,A -85,B 0,C 180,E1 -6105.217,E2 -6105.217} C_VEL
LIN {X 0,Y 495.85,Z 196.03,A -85,B 0,C 180,E1 -6108.554,E2 -6108.554} C_VEL
LIN {X 0,Y 495.871,Z 196.031,A -85,B 0,C 180,E1 -6111.852,E2 -6111.852} C_VEL
LIN {X 0,Y 495.892,Z 196.026,A -85,B 0,C 180,E1 -6114.306,E2 -6114.306} C_VEL
LIN {X 0,Y 495.989,Z 196.016,A -85,B 0,C 180,E1 -6117.563,E2 -6117.563} C_VEL
LIN {X 0,Y 495.98,Z 196.013,A -85,B 0,C 180,E1 -6120.811,E2 -6120.811} C_VEL
LIN {X 0,Y 495.988,Z 196.012,A -85,B 0,C 180,E1 -6122.436,E2 -6122.436} C_VEL
LIN {X 0,Y 495.884,Z 196.032,A -85,B 0,C 180,E1 -6125.693,E2 -6125.693} C_VEL
LIN {X 0,Y 495.834,Z 196.032,A -85,B 0,C 180,E1 -6128.148,E2 -6128.148} C_VEL
LIN {X 0,Y 495.848,Z 196.034,A -85,B 0,C 180,E1 -6131.445,E2 -6131.445} C_VEL
LIN {X 0,Y 495.787,Z 196.038,A -85,B 0,C 180,E1 -6134.783,E2 -6134.783} C_VEL
LIN {X 0,Y 495.761,Z 196.045,A -85,B 0,C 180,E1 -6137.319,E2 -6137.319} C_VEL
LIN {X 0,Y 495.767,Z 196.041,A -85,B 0,C 180,E1 -6139.89,E2 -6139.89} C_VEL
LIN {X 0,Y 495.757,Z 196.042,A -85,B 0,C 180,E1 -6142.86,E2 -6142.86} C_VEL
LIN {X 0,Y 495.777,Z 196.038,A -85,B 0,C 180,E1 -6146.068,E2 -6146.068} C_VEL
LIN {X 0,Y 495.767,Z 196.042,A -85,B 0,C 180,E1 -6148.815,E2 -6148.815} C_VEL
LIN {X 0,Y 495.752,Z 196.041,A -85,B 0,C 180,E1 -6151.725,E2 -6151.725} C_VEL
LIN {X 0,Y 495.761,Z 196.041,A -85,B 0,C 180,E1 -6154.692,E2 -6154.692} C_VEL
LIN {X 0,Y 495.727,Z 196.046,A -85,B 0,C 180,E1 -6157.561,E2 -6157.561} C_VEL
LIN {X 0,Y 495.757,Z 196.04,A -85,B 0,C 180,E1 -6160.046,E2 -6160.046} C_VEL
LIN {X 0,Y 495.715,Z 196.052,A -85,B 0,C 180,E1 -6162.884,E2 -6162.884} C_VEL
LIN {X 0,Y 495.724,Z 196.048,A -85,B 0,C 180,E1 -6165.997,E2 -6165.997} C_VEL
LIN {X 0,Y 495.735,Z 196.047,A -85,B 0,C 180,E1 -6169.296,E2 -6169.296} C_VEL
LIN {X 0,Y 495.748,Z 196.045,A -85,B 0,C 180,E1 -6171.407,E2 -6171.407} C_VEL
LIN {X 0,Y 495.746,Z 196.045,A -85,B 0,C 180,E1 -6174.461,E2 -6174.461} C_VEL
LIN {X 0,Y 495.768,Z 196.042,A -85,B 0,C 180,E1 -6177.405,E2 -6177.405} C_VEL
LIN {X 0,Y 495.763,Z 196.06,A -85,B 0,C 180,E1 -6178.387,E2 -6178.387} C_VEL
LIN {X 0,Y 501.019,Z 213.658,A -85,B 0,C 180,E1 -6180.595,E2 -6180.595} C_VEL
LIN {X 0,Y 502.304,Z 218.121,A -85,B 0,C 180,E1 -6181.137,E2 -6181.137} C_VEL
LIN {X 0,Y 501.666,Z 232.885,A -85,B 0,C 180,E1 -6182.605,E2 -6182.605} C_VEL
LIN {X 0,Y 505.342,Z 253.301,A -85,B 0,C 180,E1 -6183.144,E2 -6183.144} C_VEL
LIN {X 0,Y 503.161,Z 440.235,A -85,B 0,C 180,E1 -6185.967,E2 -6185.967} C_VEL
LIN {X 0,Y 502.673,Z 456.967,A -85,B 0,C 180,E1 -6186.38,E2 -6186.38} C_VEL
LIN {X 0,Y 502.071,Z 472.671,A -85,B 0,C 180,E1 -6186.923,E2 -6186.923} C_VEL
LIN {X 0,Y 501.443,Z 486.805,A -85,B 0,C 180,E1 -6187.546,E2 -6187.546} C_VEL
LIN {X 0,Y 500.547,Z 502.381,A -85,B 0,C 180,E1 -6188.402,E2 -6188.402} C_VEL
LIN {X 0,Y 499.667,Z 517.312,A -85,B 0,C 180,E1 -6189.411,E2 -6189.411} C_VEL
LIN {X 0,Y 498.814,Z 531.142,A -85,B 0,C 180,E1 -6190.53,E2 -6190.53} C_VEL
LIN {X 0,Y 498.039,Z 543.492,A -85,B 0,C 180,E1 -6191.7,E2 -6191.7} C_VEL
LIN {X 0,Y 497.366,Z 554.79,A -85,B 0,C 180,E1 -6192.949,E2 -6192.949} C_VEL
LIN {X 0,Y 496.691,Z 566.071,A -85,B 0,C 180,E1 -6194.403,E2 -6194.403} C_VEL
LIN {X 0,Y 496.18,Z 575.752,A -85,B 0,C 180,E1 -6195.856,E2 -6195.856} C_VEL
LIN {X 0,Y 495.801,Z 585.163,A -85,B 0,C 180,E1 -6197.514,E2 -6197.514} C_VEL
LIN {X 0,Y 495.434,Z 593.872,A -85,B 0,C 180,E1 -6199.372,E2 -6199.372} C_VEL
LIN {X 0,Y 495.165,Z 601.59,A -85,B 0,C 180,E1 -6201.428,E2 -6201.428} C_VEL
LIN {X 0,Y 495.112,Z 606.38,A -85,B 0,C 180,E1 -6203.068,E2 -6203.068} C_VEL
LIN {X 0,Y 495.035,Z 609.296,A -85,B 0,C 180,E1 -6204.295,E2 -6204.295} C_VEL
LIN {X 0,Y 494.974,Z 612.258,A -85,B 0,C 180,E1 -6205.927,E2 -6205.927} C_VEL
LIN {X 0,Y 494.991,Z 614.208,A -85,B 0,C 180,E1 -6207.557,E2 -6207.557} C_VEL
LIN {X 0,Y 494.907,Z 615.176,A -85,B 0,C 180,E1 -6209.184,E2 -6209.184} C_VEL
LIN {X 0,Y 494.906,Z 615.179,A -85,B 0,C 180,E1 -6210.812,E2 -6210.812} C_VEL
LIN {X 0,Y 494.99,Z 614.22,A -85,B 0,C 180,E1 -6212.439,E2 -6212.439} C_VEL
LIN {X 0,Y 494.973,Z 612.279,A -85,B 0,C 180,E1 -6214.069,E2 -6214.069} C_VEL
LIN {X 0,Y 495.032,Z 609.331,A -85,B 0,C 180,E1 -6215.701,E2 -6215.701} C_VEL
LIN {X 0,Y 495.136,Z 605.348,A -85,B 0,C 180,E1 -6217.337,E2 -6217.337} C_VEL
LIN {X 0,Y 495.206,Z 600.212,A -85,B 0,C 180,E1 -6218.979,E2 -6218.979} C_VEL
LIN {X 0,Y 495.444,Z 593.945,A -85,B 0,C 180,E1 -6220.624,E2 -6220.624} C_VEL
LIN {X 0,Y 495.813,Z 585.255,A -85,B 0,C 180,E1 -6222.481,E2 -6222.481} C_VEL
LIN {X 0,Y 496.176,Z 575.869,A -85,B 0,C 180,E1 -6224.14,E2 -6224.14} C_VEL
LIN {X 0,Y 496.71,Z 566.21,A -85,B 0,C 180,E1 -6225.592,E2 -6225.592} C_VEL
LIN {X 0,Y 497.367,Z 554.954,A -85,B 0,C 180,E1 -6227.047,E2 -6227.047} C_VEL
LIN {X 0,Y 498.159,Z 542.699,A -85,B 0,C 180,E1 -6228.398,E2 -6228.398} C_VEL
LIN {X 0,Y 498.974,Z 529.189,A -85,B 0,C 180,E1 -6229.657,E2 -6229.657} C_VEL
LIN {X 0,Y 499.862,Z 514.701,A -85,B 0,C 180,E1 -6230.791,E2 -6230.791} C_VEL
LIN {X 0,Y 500.682,Z 501.044,A -85,B 0,C 180,E1 -6231.687,E2 -6231.687} C_VEL
LIN {X 0,Y 501.546,Z 485.65,A -85,B 0,C 180,E1 -6232.521,E2 -6232.521} C_VEL
LIN {X 0,Y 502.212,Z 470.455,A -85,B 0,C 180,E1 -6233.175,E2 -6233.175} C_VEL
LIN {X 0,Y 502.75,Z 454.691,A -85,B 0,C 180,E1 -6233.694,E2 -6233.694} C_VEL
LIN {X 0,Y 503.28,Z 437.86,A -85,B 0,C 180,E1 -6234.078,E2 -6234.078} C_VEL
LIN {X 0,Y 505.297,Z 253.374,A -85,B 0,C 180,E1 -6236.857,E2 -6236.857} C_VEL
LIN {X 0,Y 501.718,Z 233.082,A -85,B 0,C 180,E1 -6237.394,E2 -6237.394} C_VEL
LIN {X 0,Y 502.437,Z 218.433,A -85,B 0,C 180,E1 -6238.851,E2 -6238.851} C_VEL
LIN {X 0,Y 496.872,Z 199.774,A -85,B 0,C 180,E1 -6241.153,E2 -6241.153} C_VEL
LIN {X 0,Y 495.74,Z 196.044,A -85,B 0,C 180,E1 -6241.634,E2 -6241.634} C_VEL
LIN {X 0,Y 495.763,Z 196.044,A -85,B 0,C 180,E1 -6244.54,E2 -6244.54} C_VEL
LIN {X 0,Y 495.71,Z 196.049,A -85,B 0,C 180,E1 -6247.559,E2 -6247.559} C_VEL
LIN {X 0,Y 495.745,Z 196.042,A -85,B 0,C 180,E1 -6250.697,E2 -6250.697} C_VEL
LIN {X 0,Y 495.711,Z 196.047,A -85,B 0,C 180,E1 -6253.999,E2 -6253.999} C_VEL
LIN {X 0,Y 495.733,Z 196.05,A -85,B 0,C 180,E1 -6257.118,E2 -6257.118} C_VEL
LIN {X 0,Y 495.759,Z 196.039,A -85,B 0,C 180,E1 -6259.947,E2 -6259.947} C_VEL
LIN {X 0,Y 495.703,Z 196.048,A -85,B 0,C 180,E1 -6262.551,E2 -6262.551} C_VEL
LIN {X 0,Y 495.756,Z 196.043,A -85,B 0,C 180,E1 -6265.455,E2 -6265.455} C_VEL
LIN {X 0,Y 495.729,Z 196.036,A -85,B 0,C 180,E1 -6268.362,E2 -6268.362} C_VEL
LIN {X 0,Y 495.757,Z 196.041,A -85,B 0,C 180,E1 -6271.505,E2 -6271.505} C_VEL
LIN {X 0,Y 495.759,Z 196.031,A -85,B 0,C 180,E1 -6273.931,E2 -6273.931} C_VEL
LIN {X 0,Y 495.756,Z 196.045,A -85,B 0,C 180,E1 -6277.13,E2 -6277.13} C_VEL
LIN {X 0,Y 495.746,Z 196.031,A -85,B 0,C 180,E1 -6280.109,E2 -6280.109} C_VEL
LIN {X 0,Y 495.755,Z 196.042,A -85,B 0,C 180,E1 -6282.681,E2 -6282.681} C_VEL
LIN {X 0,Y 495.756,Z 196.039,A -85,B 0,C 180,E1 -6285.217,E2 -6285.217} C_VEL
LIN {X 0,Y 495.841,Z 196.018,A -85,B 0,C 180,E1 -6288.555,E2 -6288.555} C_VEL
LIN {X 0,Y 495.839,Z 196.029,A -85,B 0,C 180,E1 -6291.852,E2 -6291.852} C_VEL
LIN {X 0,Y 495.88,Z 196.024,A -85,B 0,C 180,E1 -6294.307,E2 -6294.307} C_VEL
LIN {X 0,Y 495.958,Z 196.005,A -85,B 0,C 180,E1 -6297.564,E2 -6297.564} C_VEL
LIN {X 0,Y 495.96,Z 196.014,A -85,B 0,C 180,E1 -6300,E2 -6300} C_VEL
LIN {X 0,Y 495.959,Z 196.02,A -85,B 0,C 180,E1 -6302.437,E2 -6302.437} C_VEL
LIN {X 0,Y 495.87,Z 196.02,A -85,B 0,C 180,E1 -6305.694,E2 -6305.694} C_VEL
LIN {X 0,Y 495.84,Z 196.031,A -85,B 0,C 180,E1 -6308.149,E2 -6308.149} C_VEL
LIN {X 0,Y 495.822,Z 196.021,A -85,B 0,C 180,E1 -6311.446,E2 -6311.446} C_VEL
LIN {X 0,Y 495.762,Z 196.043,A -85,B 0,C 180,E1 -6314.784,E2 -6314.784} C_VEL
LIN {X 0,Y 495.761,Z 196.034,A -85,B 0,C 180,E1 -6317.32,E2 -6317.32} C_VEL
LIN {X 0,Y 495.748,Z 196.034,A -85,B 0,C 180,E1 -6319.892,E2 -6319.892} C_VEL
LIN {X 0,Y 495.736,Z 196.044,A -85,B 0,C 180,E1 -6322.864,E2 -6322.864} C_VEL
LIN {X 0,Y 495.763,Z 196.035,A -85,B 0,C 180,E1 -6326.07,E2 -6326.07} C_VEL
LIN {X 0,Y 495.745,Z 196.044,A -85,B 0,C 180,E1 -6328.817,E2 -6328.817} C_VEL
LIN {X 0,Y 495.729,Z 196.041,A -85,B 0,C 180,E1 -6331.728,E2 -6331.728} C_VEL
LIN {X 0,Y 495.75,Z 196.044,A -85,B 0,C 180,E1 -6334.697,E2 -6334.697} C_VEL
LIN {X 0,Y 495.707,Z 196.045,A -85,B 0,C 180,E1 -6337.564,E2 -6337.564} C_VEL
LIN {X 0,Y 495.746,Z 196.043,A -85,B 0,C 180,E1 -6340.703,E2 -6340.703} C_VEL
LIN {X 0,Y 495.708,Z 196.05,A -85,B 0,C 180,E1 -6344.005,E2 -6344.005} C_VEL
LIN {X 0,Y 495.699,Z 196.047,A -85,B 0,C 180,E1 -6347.119,E2 -6347.119} C_VEL
LIN {X 0,Y 495.743,Z 196.045,A -85,B 0,C 180,E1 -6349.956,E2 -6349.956} C_VEL
LIN {X 0,Y 495.716,Z 196.048,A -85,B 0,C 180,E1 -6352.556,E2 -6352.556} C_VEL
LIN {X 0,Y 495.769,Z 196.034,A -85,B 0,C 180,E1 -6355.46,E2 -6355.46} C_VEL
LIN {X 0,Y 495.744,Z 196.045,A -85,B 0,C 180,E1 -6358.367,E2 -6358.367} C_VEL
LIN {X 0,Y 495.727,Z 196.042,A -85,B 0,C 180,E1 -6360.793,E2 -6360.793} C_VEL
LIN {X 0,Y 495.055,Z 196.129,A -85,B 0,C 180,E1 -6361.472,E2 -6361.472} C_VEL
LIN {X 0,Y 492.182,Z 196.487,A -85,B 0,C 180,E1 -6362.574,E2 -6362.574} C_VEL
LIN {X 0,Y 489.768,Z 196.787,A -85,B 0,C 180,E1 -6363.462,E2 -6363.462} C_VEL
LIN {X 0,Y 488.755,Z 196.914,A -85,B 0,C 180,E1 -6364.148,E2 -6364.148} C_VEL
LIN {X 0,Y 488.686,Z 196.922,A -85,B 0,C 180,E1 -6364.38,E2 -6364.38} C_VEL
LIN {X 0,Y 488.716,Z 196.916,A -85,B 0,C 180,E1 -6367.156,E2 -6367.156} C_VEL
LIN {X 0,Y 488.715,Z 196.925,A -85,B 0,C 180,E1 -6369.813,E2 -6369.813} C_VEL
LIN {X 0,Y 488.679,Z 196.925,A -85,B 0,C 180,E1 -6372.424,E2 -6372.424} C_VEL
LIN {X 0,Y 488.748,Z 196.915,A -85,B 0,C 180,E1 -6375.002,E2 -6375.002} C_VEL
LIN {X 0,Y 488.806,Z 196.909,A -85,B 0,C 180,E1 -6378.39,E2 -6378.39} C_VEL
LIN {X 0,Y 488.763,Z 196.917,A -85,B 0,C 180,E1 -6381.735,E2 -6381.735} C_VEL
LIN {X 0,Y 488.816,Z 196.9,A -85,B 0,C 180,E1 -6384.226,E2 -6384.226} C_VEL
LIN {X 0,Y 488.936,Z 196.934,A -85,B 0,C 180,E1 -6387.556,E2 -6387.556} C_VEL
LIN {X 0,Y 492.026,Z 208.207,A -85,B 0,C 180,E1 -6389.096,E2 -6389.096} C_VEL
LIN {X 0,Y 498.274,Z 222.187,A -85,B 0,C 180,E1 -6389.702,E2 -6389.702} C_VEL
LIN {X 0,Y 499.123,Z 227.301,A -85,B 0,C 180,E1 -6389.835,E2 -6389.835} C_VEL
LIN {X 0,Y 496.847,Z 413.725,A -85,B 0,C 180,E1 -6392.687,E2 -6392.687} C_VEL
LIN {X 0,Y 496.36,Z 430.134,A -85,B 0,C 180,E1 -6393.096,E2 -6393.096} C_VEL
LIN {X 0,Y 495.789,Z 446.121,A -85,B 0,C 180,E1 -6393.659,E2 -6393.659} C_VEL
LIN {X 0,Y 495.115,Z 459.932,A -85,B 0,C 180,E1 -6394.276,E2 -6394.276} C_VEL
LIN {X 0,Y 494.293,Z 475.362,A -85,B 0,C 180,E1 -6395.143,E2 -6395.143} C_VEL
LIN {X 0,Y 493.353,Z 489.846,A -85,B 0,C 180,E1 -6396.135,E2 -6396.135} C_VEL
LIN {X 0,Y 492.467,Z 503.755,A -85,B 0,C 180,E1 -6397.278,E2 -6397.278} C_VEL
LIN {X 0,Y 491.661,Z 515.595,A -85,B 0,C 180,E1 -6398.415,E2 -6398.415} C_VEL
LIN {X 0,Y 490.727,Z 528.661,A -85,B 0,C 180,E1 -6399.898,E2 -6399.898} C_VEL
LIN {X 0,Y 489.982,Z 539.634,A -85,B 0,C 180,E1 -6401.376,E2 -6401.376} C_VEL
LIN {X 0,Y 489.395,Z 548.837,A -85,B 0,C 180,E1 -6402.82,E2 -6402.82} C_VEL
LIN {X 0,Y 488.973,Z 557.258,A -85,B 0,C 180,E1 -6404.357,E2 -6404.357} C_VEL
LIN {X 0,Y 488.595,Z 564.214,A -85,B 0,C 180,E1 -6405.862,E2 -6405.862} C_VEL
LIN {X 0,Y 488.306,Z 570.951,A -85,B 0,C 180,E1 -6407.594,E2 -6407.594} C_VEL
LIN {X 0,Y 488.136,Z 576.444,A -85,B 0,C 180,E1 -6409.34,E2 -6409.34} C_VEL
LIN {X 0,Y 487.919,Z 580.739,A -85,B 0,C 180,E1 -6411.108,E2 -6411.108} C_VEL
LIN {X 0,Y 487.782,Z 583.928,A -85,B 0,C 180,E1 -6412.895,E2 -6412.895} C_VEL
LIN {X 0,Y 487.766,Z 586.081,A -85,B 0,C 180,E1 -6414.804,E2 -6414.804} C_VEL
LIN {X 0,Y 487.769,Z 586.901,A -85,B 0,C 180,E1 -6416.705,E2 -6416.705} C_VEL
LIN {X 0,Y 487.825,Z 586.557,A -85,B 0,C 180,E1 -6418.499,E2 -6418.499} C_VEL
LIN {X 0,Y 487.863,Z 585.15,A -85,B 0,C 180,E1 -6420.279,E2 -6420.279} C_VEL
LIN {X 0,Y 487.885,Z 582.292,A -85,B 0,C 180,E1 -6422.208,E2 -6422.208} C_VEL
LIN {X 0,Y 488.05,Z 578.009,A -85,B 0,C 180,E1 -6424.168,E2 -6424.168} C_VEL
LIN {X 0,Y 488.268,Z 572.114,A -85,B 0,C 180,E1 -6426.168,E2 -6426.168} C_VEL
LIN {X 0,Y 488.547,Z 565.615,A -85,B 0,C 180,E1 -6427.916,E2 -6427.916} C_VEL
LIN {X 0,Y 488.974,Z 557.191,A -85,B 0,C 180,E1 -6429.762,E2 -6429.762} C_VEL
LIN {X 0,Y 489.518,Z 547.426,A -85,B 0,C 180,E1 -6431.526,E2 -6431.526} C_VEL
LIN {X 0,Y 490.176,Z 537.644,A -85,B 0,C 180,E1 -6433.01,E2 -6433.01} C_VEL
LIN {X 0,Y 490.945,Z 525.825,A -85,B 0,C 180,E1 -6434.544,E2 -6434.544} C_VEL
LIN {X 0,Y 491.818,Z 513.54,A -85,B 0,C 180,E1 -6435.895,E2 -6435.895} C_VEL
LIN {X 0,Y 492.726,Z 500.455,A -85,B 0,C 180,E1 -6437.12,E2 -6437.12} C_VEL
LIN {X 0,Y 493.683,Z 485.907,A -85,B 0,C 180,E1 -6438.257,E2 -6438.257} C_VEL
LIN {X 0,Y 494.535,Z 471.704,A -85,B 0,C 180,E1 -6439.177,E2 -6439.177} C_VEL
LIN {X 0,Y 495.329,Z 455.953,A -85,B 0,C 180,E1 -6440.013,E2 -6440.013} C_VEL
LIN {X 0,Y 496.036,Z 439.859,A -85,B 0,C 180,E1 -6440.681,E2 -6440.681} C_VEL
LIN {X 0,Y 496.62,Z 423.719,A -85,B 0,C 180,E1 -6441.181,E2 -6441.181} C_VEL
LIN {X 0,Y 496.999,Z 406.773,A -85,B 0,C 180,E1 -6441.529,E2 -6441.529} C_VEL
LIN {X 0,Y 499.259,Z 226.566,A -85,B 0,C 180,E1 -6444.279,E2 -6444.279} C_VEL
LIN {X 0,Y 497.942,Z 221.047,A -85,B 0,C 180,E1 -6444.448,E2 -6444.448} C_VEL
LIN {X 0,Y 492.105,Z 208.324,A -85,B 0,C 180,E1 -6445.046,E2 -6445.046} C_VEL
LIN {X 0,Y 488.754,Z 196.917,A -85,B 0,C 180,E1 -6446.663,E2 -6446.663} C_VEL
LIN {X 0,Y 488.726,Z 196.919,A -85,B 0,C 180,E1 -6449.78,E2 -6449.78} C_VEL
LIN {X 0,Y 488.794,Z 196.91,A -85,B 0,C 180,E1 -6453.056,E2 -6453.056} C_VEL
LIN {X 0,Y 488.681,Z 196.925,A -85,B 0,C 180,E1 -6456.253,E2 -6456.253} C_VEL
LIN {X 0,Y 488.747,Z 196.912,A -85,B 0,C 180,E1 -6459.175,E2 -6459.175} C_VEL
LIN {X 0,Y 488.734,Z 196.913,A -85,B 0,C 180,E1 -6462.423,E2 -6462.423} C_VEL
LIN {X 0,Y 488.762,Z 196.912,A -85,B 0,C 180,E1 -6464.999,E2 -6464.999} C_VEL
LIN {X 0,Y 488.804,Z 196.909,A -85,B 0,C 180,E1 -6468.387,E2 -6468.387} C_VEL
LIN {X 0,Y 488.814,Z 196.91,A -85,B 0,C 180,E1 -6471.733,E2 -6471.733} C_VEL
LIN {X 0,Y 488.851,Z 196.904,A -85,B 0,C 180,E1 -6474.224,E2 -6474.224} C_VEL
LIN {X 0,Y 488.957,Z 196.891,A -85,B 0,C 180,E1 -6477.528,E2 -6477.528} C_VEL
LIN {X 0,Y 488.932,Z 196.891,A -85,B 0,C 180,E1 -6480.823,E2 -6480.823} C_VEL
LIN {X 0,Y 488.956,Z 196.888,A -85,B 0,C 180,E1 -6482.471,E2 -6482.471} C_VEL
LIN {X 0,Y 488.843,Z 196.908,A -85,B 0,C 180,E1 -6485.775,E2 -6485.775} C_VEL
LIN {X 0,Y 488.783,Z 196.91,A -85,B 0,C 180,E1 -6488.267,E2 -6488.267} C_VEL
LIN {X 0,Y 488.803,Z 196.913,A -85,B 0,C 180,E1 -6491.612,E2 -6491.612} C_VEL
LIN {X 0,Y 488.759,Z 196.915,A -85,B 0,C 180,E1 -6495,E2 -6495} C_VEL
LIN {X 0,Y 488.745,Z 196.913,A -85,B 0,C 180,E1 -6498.442,E2 -6498.442} C_VEL
LIN {X 0,Y 488.704,Z 196.924,A -85,B 0,C 180,E1 -6501.07,E2 -6501.07} C_VEL
LIN {X 0,Y 488.673,Z 196.923,A -85,B 0,C 180,E1 -6503.746,E2 -6503.746} C_VEL
LIN {X 0,Y 488.79,Z 196.912,A -85,B 0,C 180,E1 -6506.943,E2 -6506.943} C_VEL
LIN {X 0,Y 488.707,Z 196.918,A -85,B 0,C 180,E1 -6510.362,E2 -6510.362} C_VEL
LIN {X 0,Y 488.709,Z 196.921,A -85,B 0,C 180,E1 -6513.479,E2 -6513.479} C_VEL
LIN {X 0,Y 488.681,Z 196.922,A -85,B 0,C 180,E1 -6516.354,E2 -6516.354} C_VEL
LIN {X 0,Y 488.7,Z 196.925,A -85,B 0,C 180,E1 -6519.254,E2 -6519.254} C_VEL
LIN {X 0,Y 488.697,Z 196.92,A -85,B 0,C 180,E1 -6521.598,E2 -6521.598} C_VEL
LIN {X 0,Y 488.701,Z 196.921,A -85,B 0,C 180,E1 -6524.802,E2 -6524.802} C_VEL
LIN {X 0,Y 488.667,Z 196.924,A -85,B 0,C 180,E1 -6527.471,E2 -6527.471} C_VEL
LIN {X 0,Y 488.697,Z 196.923,A -85,B 0,C 180,E1 -6530.745,E2 -6530.745} C_VEL
LIN {X 0,Y 488.67,Z 196.926,A -85,B 0,C 180,E1 -6533.866,E2 -6533.866} C_VEL
LIN {X 0,Y 488.74,Z 196.921,A -85,B 0,C 180,E1 -6536.876,E2 -6536.876} C_VEL
LIN {X 0,Y 488.733,Z 197.053,A -85,B 0,C 180,E1 -6538.003,E2 -6538.003} C_VEL
LIN {X 0,Y 494.163,Z 214.92,A -85,B 0,C 180,E1 -6540.299,E2 -6540.299} C_VEL
LIN {X 0,Y 495.734,Z 220.525,A -85,B 0,C 180,E1 -6540.987,E2 -6540.987} C_VEL
LIN {X 0,Y 495.092,Z 232.447,A -85,B 0,C 180,E1 -6542.193,E2 -6542.193} C_VEL
LIN {X 0,Y 498.99,Z 254.909,A -85,B 0,C 180,E1 -6542.8,E2 -6542.8} C_VEL
LIN {X 0,Y 496.703,Z 438.631,A -85,B 0,C 180,E1 -6545.611,E2 -6545.611} C_VEL
LIN {X 0,Y 496.16,Z 454.829,A -85,B 0,C 180,E1 -6545.995,E2 -6545.995} C_VEL
LIN {X 0,Y 495.6,Z 471.079,A -85,B 0,C 180,E1 -6546.549,E2 -6546.549} C_VEL
LIN {X 0,Y 494.837,Z 485.464,A -85,B 0,C 180,E1 -6547.174,E2 -6547.174} C_VEL
LIN {X 0,Y 493.984,Z 500.959,A -85,B 0,C 180,E1 -6548.03,E2 -6548.03} C_VEL
LIN {X 0,Y 493.157,Z 514.169,A -85,B 0,C 180,E1 -6548.908,E2 -6548.908} C_VEL
LIN {X 0,Y 492.258,Z 527.624,A -85,B 0,C 180,E1 -6549.96,E2 -6549.96} C_VEL
LIN {X 0,Y 491.303,Z 541.192,A -85,B 0,C 180,E1 -6551.223,E2 -6551.223} C_VEL
LIN {X 0,Y 490.564,Z 552.74,A -85,B 0,C 180,E1 -6552.49,E2 -6552.49} C_VEL
LIN {X 0,Y 489.806,Z 564.701,A -85,B 0,C 180,E1 -6554.018,E2 -6554.018} C_VEL
LIN {X 0,Y 489.271,Z 574.264,A -85,B 0,C 180,E1 -6555.44,E2 -6555.44} C_VEL
LIN {X 0,Y 488.77,Z 583.816,A -85,B 0,C 180,E1 -6557.121,E2 -6557.121} C_VEL
LIN {X 0,Y 488.437,Z 591.815,A -85,B 0,C 180,E1 -6558.798,E2 -6558.798} C_VEL
LIN {X 0,Y 488.134,Z 598.488,A -85,B 0,C 180,E1 -6560.468,E2 -6560.468} C_VEL
LIN {X 0,Y 488.047,Z 603.901,A -85,B 0,C 180,E1 -6562.135,E2 -6562.135} C_VEL
LIN {X 0,Y 488.001,Z 607.676,A -85,B 0,C 180,E1 -6563.568,E2 -6563.568} C_VEL
LIN {X 0,Y 487.907,Z 610.682,A -85,B 0,C 180,E1 -6565.04,E2 -6565.04} C_VEL
LIN {X 0,Y 487.942,Z 613.184,A -85,B 0,C 180,E1 -6566.695,E2 -6566.695} C_VEL
LIN {X 0,Y 487.885,Z 614.594,A -85,B 0,C 180,E1 -6568.347,E2 -6568.347} C_VEL
LIN {X 0,Y 487.814,Z 615.128,A -85,B 0,C 180,E1 -6569.998,E2 -6569.998} C_VEL
LIN {X 0,Y 487.885,Z 614.604,A -85,B 0,C 180,E1 -6571.649,E2 -6571.649} C_VEL
LIN {X 0,Y 487.941,Z 613.204,A -85,B 0,C 180,E1 -6573.301,E2 -6573.301} C_VEL
LIN {X 0,Y 487.906,Z 610.716,A -85,B 0,C 180,E1 -6574.956,E2 -6574.956} C_VEL
LIN {X 0,Y 487.991,Z 607.295,A -85,B 0,C 180,E1 -6576.614,E2 -6576.614} C_VEL
LIN {X 0,Y 488.091,Z 601.438,A -85,B 0,C 180,E1 -6578.693,E2 -6578.693} C_VEL
LIN {X 0,Y 488.38,Z 593.733,A -85,B 0,C 180,E1 -6580.78,E2 -6580.78} C_VEL
LIN {X 0,Y 488.77,Z 585.04,A -85,B 0,C 180,E1 -6582.664,E2 -6582.664} C_VEL
LIN {X 0,Y 489.168,Z 575.649,A -85,B 0,C 180,E1 -6584.347,E2 -6584.347} C_VEL
LIN {X 0,Y 489.751,Z 565.986,A -85,B 0,C 180,E1 -6585.819,E2 -6585.819} C_VEL
LIN {X 0,Y 490.455,Z 554.724,A -85,B 0,C 180,E1 -6587.295,E2 -6587.295} C_VEL
LIN {X 0,Y 491.295,Z 542.465,A -85,B 0,C 180,E1 -6588.665,E2 -6588.665} C_VEL
LIN {X 0,Y 492.218,Z 529.072,A -85,B 0,C 180,E1 -6589.927,E2 -6589.927} C_VEL
LIN {X 0,Y 493.051,Z 515.88,A -85,B 0,C 180,E1 -6590.983,E2 -6590.983} C_VEL
LIN {X 0,Y 493.999,Z 501.162,A -85,B 0,C 180,E1 -6591.972,E2 -6591.972} C_VEL
LIN {X 0,Y 494.92,Z 485.805,A -85,B 0,C 180,E1 -6592.817,E2 -6592.817} C_VEL
LIN {X 0,Y 495.703,Z 468.846,A -85,B 0,C 180,E1 -6593.552,E2 -6593.552} C_VEL
LIN {X 0,Y 496.298,Z 452.512,A -85,B 0,C 180,E1 -6594.077,E2 -6594.077} C_VEL
LIN {X 0,Y 496.799,Z 436.025,A -85,B 0,C 180,E1 -6594.438,E2 -6594.438} C_VEL
LIN {X 0,Y 498.96,Z 254.809,A -85,B 0,C 180,E1 -6597.198,E2 -6597.198} C_VEL
LIN {X 0,Y 495.141,Z 232.905,A -85,B 0,C 180,E1 -6597.784,E2 -6597.784} C_VEL
LIN {X 0,Y 495.808,Z 220.747,A -85,B 0,C 180,E1 -6599.008,E2 -6599.008} C_VEL
LIN {X 0,Y 490.847,Z 203.861,A -85,B 0,C 180,E1 -6601.114,E2 -6601.114} C_VEL
LIN {X 0,Y 488.703,Z 196.913,A -85,B 0,C 180,E1 -6602.043,E2 -6602.043} C_VEL
LIN {X 0,Y 488.7,Z 196.924,A -85,B 0,C 180,E1 -6605.112,E2 -6605.112} C_VEL
LIN {X 0,Y 488.66,Z 196.926,A -85,B 0,C 180,E1 -6608.198,E2 -6608.198} C_VEL
LIN {X 0,Y 488.697,Z 196.918,A -85,B 0,C 180,E1 -6610.342,E2 -6610.342} C_VEL
LIN {X 0,Y 488.664,Z 196.927,A -85,B 0,C 180,E1 -6613.652,E2 -6613.652} C_VEL
LIN {X 0,Y 488.668,Z 196.921,A -85,B 0,C 180,E1 -6616.344,E2 -6616.344} C_VEL
LIN {X 0,Y 488.724,Z 196.917,A -85,B 0,C 180,E1 -6619.649,E2 -6619.649} C_VEL
LIN {X 0,Y 488.655,Z 196.926,A -85,B 0,C 180,E1 -6622.839,E2 -6622.839} C_VEL
LIN {X 0,Y 488.706,Z 196.919,A -85,B 0,C 180,E1 -6625.886,E2 -6625.886} C_VEL
LIN {X 0,Y 488.664,Z 196.92,A -85,B 0,C 180,E1 -6628.819,E2 -6628.819} C_VEL
LIN {X 0,Y 488.714,Z 196.917,A -85,B 0,C 180,E1 -6631.67,E2 -6631.67} C_VEL
LIN {X 0,Y 488.716,Z 196.91,A -85,B 0,C 180,E1 -6634.443,E2 -6634.443} C_VEL
LIN {X 0,Y 488.717,Z 196.922,A -85,B 0,C 180,E1 -6637.153,E2 -6637.153} C_VEL
LIN {X 0,Y 488.697,Z 196.909,A -85,B 0,C 180,E1 -6639.81,E2 -6639.81} C_VEL
LIN {X 0,Y 488.702,Z 196.917,A -85,B 0,C 180,E1 -6642.423,E2 -6642.423} C_VEL
LIN {X 0,Y 488.728,Z 196.918,A -85,B 0,C 180,E1 -6644.999,E2 -6644.999} C_VEL
LIN {X 0,Y 488.8,Z 196.892,A -85,B 0,C 180,E1 -6648.388,E2 -6648.388} C_VEL
LIN {X 0,Y 488.784,Z 196.908,A -85,B 0,C 180,E1 -6651.733,E2 -6651.733} C_VEL
LIN {X 0,Y 488.836,Z 196.901,A -85,B 0,C 180,E1 -6654.224,E2 -6654.224} C_VEL
LIN {X 0,Y 488.927,Z 196.881,A -85,B 0,C 180,E1 -6657.529,E2 -6657.529} C_VEL
LIN {X 0,Y 488.932,Z 196.889,A -85,B 0,C 180,E1 -6660,E2 -6660} C_VEL
LIN {X 0,Y 488.927,Z 196.896,A -85,B 0,C 180,E1 -6662.472,E2 -6662.472} C_VEL
LIN {X 0,Y 488.828,Z 196.897,A -85,B 0,C 180,E1 -6665.777,E2 -6665.777} C_VEL
LIN {X 0,Y 488.785,Z 196.911,A -85,B 0,C 180,E1 -6668.267,E2 -6668.267} C_VEL
LIN {X 0,Y 488.775,Z 196.898,A -85,B 0,C 180,E1 -6671.614,E2 -6671.614} C_VEL
LIN {X 0,Y 488.733,Z 196.916,A -85,B 0,C 180,E1 -6675.002,E2 -6675.002} C_VEL
LIN {X 0,Y 488.724,Z 196.912,A -85,B 0,C 180,E1 -6678.444,E2 -6678.444} C_VEL
LIN {X 0,Y 488.683,Z 196.921,A -85,B 0,C 180,E1 -6681.072,E2 -6681.072} C_VEL
LIN {X 0,Y 488.672,Z 196.922,A -85,B 0,C 180,E1 -6683.747,E2 -6683.747} C_VEL
LIN {X 0,Y 488.764,Z 196.909,A -85,B 0,C 180,E1 -6686.946,E2 -6686.946} C_VEL
LIN {X 0,Y 488.683,Z 196.927,A -85,B 0,C 180,E1 -6690.365,E2 -6690.365} C_VEL
LIN {X 0,Y 488.71,Z 196.91,A -85,B 0,C 180,E1 -6693.487,E2 -6693.487} C_VEL
LIN {X 0,Y 488.664,Z 196.93,A -85,B 0,C 180,E1 -6696.358,E2 -6696.358} C_VEL
LIN {X 0,Y 488.677,Z 196.912,A -85,B 0,C 180,E1 -6699.257,E2 -6699.257} C_VEL
LIN {X 0,Y 488.688,Z 196.921,A -85,B 0,C 180,E1 -6701.603,E2 -6701.603} C_VEL
LIN {X 0,Y 488.682,Z 196.915,A -85,B 0,C 180,E1 -6704.806,E2 -6704.806} C_VEL
LIN {X 0,Y 488.671,Z 196.923,A -85,B 0,C 180,E1 -6707.477,E2 -6707.477} C_VEL
LIN {X 0,Y 488.685,Z 196.918,A -85,B 0,C 180,E1 -6710.749,E2 -6710.749} C_VEL
LIN {X 0,Y 488.67,Z 196.928,A -85,B 0,C 180,E1 -6713.871,E2 -6713.871} C_VEL
LIN {X 0,Y 488.727,Z 196.916,A -85,B 0,C 180,E1 -6716.88,E2 -6716.88} C_VEL
LIN {X 0,Y 488.713,Z 196.92,A -85,B 0,C 180,E1 -6719.784,E2 -6719.784} C_VEL
LIN {X 0,Y 488.706,Z 196.918,A -85,B 0,C 180,E1 -6723.078,E2 -6723.078} C_VEL
LIN {X 0,Y 488.686,Z 196.922,A -85,B 0,C 180,E1 -6724.38,E2 -6724.38} C_VEL
LIN {X 0,Y 488.051,Z 197.005,A -85,B 0,C 180,E1 -6725.068,E2 -6725.068} C_VEL
LIN {X 0,Y 485.2,Z 197.361,A -85,B 0,C 180,E1 -6726.186,E2 -6726.186} C_VEL
LIN {X 0,Y 482.766,Z 197.661,A -85,B 0,C 180,E1 -6727.087,E2 -6727.087} C_VEL
LIN {X 0,Y 481.715,Z 197.791,A -85,B 0,C 180,E1 -6727.782,E2 -6727.782} C_VEL
LIN {X 0,Y 481.628,Z 197.8,A -85,B 0,C 180,E1 -6728.018,E2 -6728.018} C_VEL
LIN {X 0,Y 481.692,Z 197.793,A -85,B 0,C 180,E1 -6730.395,E2 -6730.395} C_VEL
LIN {X 0,Y 481.619,Z 197.802,A -85,B 0,C 180,E1 -6733.034,E2 -6733.034} C_VEL
LIN {X 0,Y 481.677,Z 197.8,A -85,B 0,C 180,E1 -6735.641,E2 -6735.641} C_VEL
LIN {X 0,Y 481.751,Z 197.788,A -85,B 0,C 180,E1 -6738.218,E2 -6738.218} C_VEL
LIN {X 0,Y 481.722,Z 197.795,A -85,B 0,C 180,E1 -6741.613,E2 -6741.613} C_VEL
LIN {X 0,Y 481.778,Z 197.777,A -85,B 0,C 180,E1 -6744.141,E2 -6744.141} C_VEL
LIN {X 0,Y 481.817,Z 197.911,A -85,B 0,C 180,E1 -6747.18,E2 -6747.18} C_VEL
LIN {X 0,Y 484.871,Z 208.539,A -85,B 0,C 180,E1 -6748.654,E2 -6748.654} C_VEL
LIN {X 0,Y 492.304,Z 224.938,A -85,B 0,C 180,E1 -6749.388,E2 -6749.388} C_VEL
LIN {X 0,Y 492.804,Z 227.852,A -85,B 0,C 180,E1 -6749.465,E2 -6749.465} C_VEL
LIN {X 0,Y 490.373,Z 414.557,A -85,B 0,C 180,E1 -6752.363,E2 -6752.363} C_VEL
LIN {X 0,Y 489.859,Z 430.739,A -85,B 0,C 180,E1 -6752.777,E2 -6752.777} C_VEL
LIN {X 0,Y 489.236,Z 446.643,A -85,B 0,C 180,E1 -6753.347,E2 -6753.347} C_VEL
LIN {X 0,Y 488.468,Z 461.363,A -85,B 0,C 180,E1 -6754.024,E2 -6754.024} C_VEL
LIN {X 0,Y 487.66,Z 475.931,A -85,B 0,C 180,E1 -6754.859,E2 -6754.859} C_VEL
LIN {X 0,Y 486.635,Z 490.943,A -85,B 0,C 180,E1 -6755.908,E2 -6755.908} C_VEL
LIN {X 0,Y 485.664,Z 504.724,A -85,B 0,C 180,E1 -6757.067,E2 -6757.067} C_VEL
LIN {X 0,Y 484.732,Z 517.515,A -85,B 0,C 180,E1 -6758.338,E2 -6758.338} C_VEL
LIN {X 0,Y 483.934,Z 528.209,A -85,B 0,C 180,E1 -6759.573,E2 -6759.573} C_VEL
LIN {X 0,Y 483.096,Z 539.588,A -85,B 0,C 180,E1 -6761.115,E2 -6761.115} C_VEL
LIN {X 0,Y 482.437,Z 549.084,A -85,B 0,C 180,E1 -6762.623,E2 -6762.623} C_VEL
LIN {X 0,Y 481.92,Z 558.334,A -85,B 0,C 180,E1 -6764.356,E2 -6764.356} C_VEL
LIN {X 0,Y 481.474,Z 566.118,A -85,B 0,C 180,E1 -6766.103,E2 -6766.103} C_VEL
LIN {X 0,Y 481.176,Z 572.51,A -85,B 0,C 180,E1 -6767.863,E2 -6767.863} C_VEL
LIN {X 0,Y 481.02,Z 577.714,A -85,B 0,C 180,E1 -6769.637,E2 -6769.637} C_VEL
LIN {X 0,Y 480.809,Z 581.805,A -85,B 0,C 180,E1 -6771.435,E2 -6771.435} C_VEL
LIN {X 0,Y 480.662,Z 584.687,A -85,B 0,C 180,E1 -6773.253,E2 -6773.253} C_VEL
LIN {X 0,Y 480.659,Z 586.482,A -85,B 0,C 180,E1 -6775.09,E2 -6775.09} C_VEL
LIN {X 0,Y 480.667,Z 587.153,A -85,B 0,C 180,E1 -6776.954,E2 -6776.954} C_VEL
LIN {X 0,Y 480.72,Z 586.58,A -85,B 0,C 180,E1 -6778.847,E2 -6778.847} C_VEL
LIN {X 0,Y 480.76,Z 584.791,A -85,B 0,C 180,E1 -6780.775,E2 -6780.775} C_VEL
LIN {X 0,Y 480.82,Z 581.665,A -85,B 0,C 180,E1 -6782.74,E2 -6782.74} C_VEL
LIN {X 0,Y 480.968,Z 578.308,A -85,B 0,C 180,E1 -6784.235,E2 -6784.235} C_VEL
LIN {X 0,Y 481.211,Z 572.813,A -85,B 0,C 180,E1 -6786.153,E2 -6786.153} C_VEL
LIN {X 0,Y 481.515,Z 566.199,A -85,B 0,C 180,E1 -6787.985,E2 -6787.985} C_VEL
LIN {X 0,Y 481.969,Z 557.585,A -85,B 0,C 180,E1 -6789.912,E2 -6789.912} C_VEL
LIN {X 0,Y 482.593,Z 547.392,A -85,B 0,C 180,E1 -6791.779,E2 -6791.779} C_VEL
LIN {X 0,Y 483.461,Z 535.967,A -85,B 0,C 180,E1 -6793.513,E2 -6793.513} C_VEL
LIN {X 0,Y 484.188,Z 524.907,A -85,B 0,C 180,E1 -6794.933,E2 -6794.933} C_VEL
LIN {X 0,Y 485.098,Z 512.975,A -85,B 0,C 180,E1 -6796.244,E2 -6796.244} C_VEL
LIN {X 0,Y 486.107,Z 499.48,A -85,B 0,C 180,E1 -6797.506,E2 -6797.506} C_VEL
LIN {X 0,Y 487.082,Z 485.346,A -85,B 0,C 180,E1 -6798.617,E2 -6798.617} C_VEL
LIN {X 0,Y 488.052,Z 469.966,A -85,B 0,C 180,E1 -6799.608,E2 -6799.608} C_VEL
LIN {X 0,Y 488.818,Z 455.597,A -85,B 0,C 180,E1 -6800.363,E2 -6800.363} C_VEL
LIN {X 0,Y 489.585,Z 439.142,A -85,B 0,C 180,E1 -6801.045,E2 -6801.045} C_VEL
LIN {X 0,Y 490.219,Z 422.634,A -85,B 0,C 180,E1 -6801.548,E2 -6801.548} C_VEL
LIN {X 0,Y 490.603,Z 405.835,A -85,B 0,C 180,E1 -6801.89,E2 -6801.89} C_VEL
LIN {X 0,Y 492.917,Z 227.661,A -85,B 0,C 180,E1 -6804.649,E2 -6804.649} C_VEL
LIN {X 0,Y 492.002,Z 223.985,A -85,B 0,C 180,E1 -6804.767,E2 -6804.767} C_VEL
LIN {X 0,Y 484.917,Z 208.74,A -85,B 0,C 180,E1 -6805.486,E2 -6805.486} C_VEL
LIN {X 0,Y 481.671,Z 197.801,A -85,B 0,C 180,E1 -6807.077,E2 -6807.077} C_VEL
LIN {X 0,Y 481.681,Z 197.799,A -85,B 0,C 180,E1 -6810.259,E2 -6810.259} C_VEL
LIN {X 0,Y 481.747,Z 197.788,A -85,B 0,C 180,E1 -6813.112,E2 -6813.112} C_VEL
LIN {X 0,Y 481.662,Z 197.801,A -85,B 0,C 180,E1 -6815.886,E2 -6815.886} C_VEL
LIN {X 0,Y 481.704,Z 197.789,A -85,B 0,C 180,E1 -6819.027,E2 -6819.027} C_VEL
LIN {X 0,Y 481.707,Z 197.79,A -85,B 0,C 180,E1 -6822.158,E2 -6822.158} C_VEL
LIN {X 0,Y 481.743,Z 197.786,A -85,B 0,C 180,E1 -6824.775,E2 -6824.775} C_VEL
LIN {X 0,Y 481.75,Z 197.79,A -85,B 0,C 180,E1 -6828.215,E2 -6828.215} C_VEL
LIN {X 0,Y 481.76,Z 197.788,A -85,B 0,C 180,E1 -6831.611,E2 -6831.611} C_VEL
LIN {X 0,Y 481.813,Z 197.782,A -85,B 0,C 180,E1 -6834.139,E2 -6834.139} C_VEL
LIN {X 0,Y 481.924,Z 197.767,A -85,B 0,C 180,E1 -6837.492,E2 -6837.492} C_VEL
LIN {X 0,Y 481.883,Z 197.769,A -85,B 0,C 180,E1 -6840.835,E2 -6840.835} C_VEL
LIN {X 0,Y 481.923,Z 197.764,A -85,B 0,C 180,E1 -6842.507,E2 -6842.507} C_VEL
LIN {X 0,Y 481.804,Z 197.783,A -85,B 0,C 180,E1 -6845.86,E2 -6845.86} C_VEL
LIN {X 0,Y 481.738,Z 197.787,A -85,B 0,C 180,E1 -6848.388,E2 -6848.388} C_VEL
LIN {X 0,Y 481.748,Z 197.789,A -85,B 0,C 180,E1 -6851.785,E2 -6851.785} C_VEL
LIN {X 0,Y 481.74,Z 197.792,A -85,B 0,C 180,E1 -6855.224,E2 -6855.224} C_VEL
LIN {X 0,Y 481.706,Z 197.79,A -85,B 0,C 180,E1 -6858.722,E2 -6858.722} C_VEL
LIN {X 0,Y 481.643,Z 197.802,A -85,B 0,C 180,E1 -6861.394,E2 -6861.394} C_VEL
LIN {X 0,Y 481.655,Z 197.795,A -85,B 0,C 180,E1 -6864.114,E2 -6864.114} C_VEL
LIN {X 0,Y 481.744,Z 197.79,A -85,B 0,C 180,E1 -6867.138,E2 -6867.138} C_VEL
LIN {X 0,Y 481.676,Z 197.796,A -85,B 0,C 180,E1 -6869.741,E2 -6869.741} C_VEL
LIN {X 0,Y 481.651,Z 197.798,A -85,B 0,C 180,E1 -6872.675,E2 -6872.675} C_VEL
LIN {X 0,Y 481.634,Z 197.801,A -85,B 0,C 180,E1 -6875.709,E2 -6875.709} C_VEL
LIN {X 0,Y 481.669,Z 197.799,A -85,B 0,C 180,E1 -6878.859,E2 -6878.859} C_VEL
LIN {X 0,Y 481.646,Z 197.798,A -85,B 0,C 180,E1 -6881.911,E2 -6881.911} C_VEL
LIN {X 0,Y 481.654,Z 197.799,A -85,B 0,C 180,E1 -6884.458,E2 -6884.458} C_VEL
LIN {X 0,Y 481.629,Z 197.8,A -85,B 0,C 180,E1 -6887.837,E2 -6887.837} C_VEL
LIN {X 0,Y 481.668,Z 197.803,A -85,B 0,C 180,E1 -6891.14,E2 -6891.14} C_VEL
LIN {X 0,Y 481.661,Z 197.8,A -85,B 0,C 180,E1 -6894.795,E2 -6894.795} C_VEL
LIN {X 0,Y 481.688,Z 197.932,A -85,B 0,C 180,E1 -6897.589,E2 -6897.589} C_VEL
LIN {X 0,Y 487.192,Z 215.814,A -85,B 0,C 180,E1 -6899.943,E2 -6899.943} C_VEL
LIN {X 0,Y 488.98,Z 222.203,A -85,B 0,C 180,E1 -6900.746,E2 -6900.746} C_VEL
LIN {X 0,Y 488.89,Z 227.192,A -85,B 0,C 180,E1 -6901.27,E2 -6901.27} C_VEL
LIN {X 0,Y 488.601,Z 232.427,A -85,B 0,C 180,E1 -6901.797,E2 -6901.797} C_VEL
LIN {X 0,Y 492.667,Z 255.68,A -85,B 0,C 180,E1 -6902.435,E2 -6902.435} C_VEL
LIN {X 0,Y 490.248,Z 438.646,A -85,B 0,C 180,E1 -6905.274,E2 -6905.274} C_VEL
LIN {X 0,Y 489.635,Z 455.465,A -85,B 0,C 180,E1 -6905.683,E2 -6905.683} C_VEL
LIN {X 0,Y 488.99,Z 472.107,A -85,B 0,C 180,E1 -6906.269,E2 -6906.269} C_VEL
LIN {X 0,Y 488.199,Z 486.249,A -85,B 0,C 180,E1 -6906.902,E2 -6906.902} C_VEL
LIN {X 0,Y 487.248,Z 502.339,A -85,B 0,C 180,E1 -6907.813,E2 -6907.813} C_VEL
LIN {X 0,Y 486.357,Z 515.349,A -85,B 0,C 180,E1 -6908.71,E2 -6908.71} C_VEL
LIN {X 0,Y 485.405,Z 528.554,A -85,B 0,C 180,E1 -6909.776,E2 -6909.776} C_VEL
LIN {X 0,Y 484.399,Z 541.997,A -85,B 0,C 180,E1 -6911.055,E2 -6911.055} C_VEL
LIN {X 0,Y 483.56,Z 554.292,A -85,B 0,C 180,E1 -6912.446,E2 -6912.446} C_VEL
LIN {X 0,Y 482.791,Z 565.587,A -85,B 0,C 180,E1 -6913.942,E2 -6913.942} C_VEL
LIN {X 0,Y 482.206,Z 575.282,A -85,B 0,C 180,E1 -6915.437,E2 -6915.437} C_VEL
LIN {X 0,Y 481.721,Z 584.701,A -85,B 0,C 180,E1 -6917.143,E2 -6917.143} C_VEL
LIN {X 0,Y 481.407,Z 591.59,A -85,B 0,C 180,E1 -6918.632,E2 -6918.632} C_VEL
LIN {X 0,Y 481.066,Z 598.267,A -85,B 0,C 180,E1 -6920.326,E2 -6920.326} C_VEL
LIN {X 0,Y 480.954,Z 603.684,A -85,B 0,C 180,E1 -6922.019,E2 -6922.019} C_VEL
LIN {X 0,Y 480.912,Z 607.704,A -85,B 0,C 180,E1 -6923.585,E2 -6923.585} C_VEL
LIN {X 0,Y 480.832,Z 610.472,A -85,B 0,C 180,E1 -6924.967,E2 -6924.967} C_VEL
LIN {X 0,Y 480.846,Z 612.976,A -85,B 0,C 180,E1 -6926.646,E2 -6926.646} C_VEL
LIN {X 0,Y 480.816,Z 614.389,A -85,B 0,C 180,E1 -6928.323,E2 -6928.323} C_VEL
LIN {X 0,Y 480.738,Z 614.924,A -85,B 0,C 180,E1 -6929.998,E2 -6929.998} C_VEL
LIN {X 0,Y 480.815,Z 614.401,A -85,B 0,C 180,E1 -6931.673,E2 -6931.673} C_VEL
LIN {X 0,Y 480.845,Z 612.999,A -85,B 0,C 180,E1 -6933.349,E2 -6933.349} C_VEL
LIN {X 0,Y 480.831,Z 610.511,A -85,B 0,C 180,E1 -6935.029,E2 -6935.029} C_VEL
LIN {X 0,Y 480.901,Z 607.089,A -85,B 0,C 180,E1 -6936.712,E2 -6936.712} C_VEL
LIN {X 0,Y 481.03,Z 601.229,A -85,B 0,C 180,E1 -6938.822,E2 -6938.822} C_VEL
LIN {X 0,Y 481.312,Z 593.52,A -85,B 0,C 180,E1 -6940.94,E2 -6940.94} C_VEL
LIN {X 0,Y 481.724,Z 584.824,A -85,B 0,C 180,E1 -6942.853,E2 -6942.853} C_VEL
LIN {X 0,Y 482.205,Z 575.431,A -85,B 0,C 180,E1 -6944.559,E2 -6944.559} C_VEL
LIN {X 0,Y 482.869,Z 565.172,A -85,B 0,C 180,E1 -6946.136,E2 -6946.136} C_VEL
LIN {X 0,Y 483.561,Z 554.49,A -85,B 0,C 180,E1 -6947.55,E2 -6947.55} C_VEL
LIN {X 0,Y 484.465,Z 542.224,A -85,B 0,C 180,E1 -6948.938,E2 -6948.938} C_VEL
LIN {X 0,Y 485.426,Z 528.921,A -85,B 0,C 180,E1 -6950.208,E2 -6950.208} C_VEL
LIN {X 0,Y 486.344,Z 515.62,A -85,B 0,C 180,E1 -6951.286,E2 -6951.286} C_VEL
LIN {X 0,Y 487.339,Z 501.271,A -85,B 0,C 180,E1 -6952.264,E2 -6952.264} C_VEL
LIN {X 0,Y 488.123,Z 488.544,A -85,B 0,C 180,E1 -6952.985,E2 -6952.985} C_VEL
LIN {X 0,Y 488.97,Z 472.426,A -85,B 0,C 180,E1 -6953.728,E2 -6953.728} C_VEL
LIN {X 0,Y 489.657,Z 455.789,A -85,B 0,C 180,E1 -6954.312,E2 -6954.312} C_VEL
LIN {X 0,Y 490.262,Z 440.294,A -85,B 0,C 180,E1 -6954.695,E2 -6954.695} C_VEL
LIN {X 0,Y 492.613,Z 255.556,A -85,B 0,C 180,E1 -6957.559,E2 -6957.559} C_VEL
LIN {X 0,Y 488.557,Z 232.786,A -85,B 0,C 180,E1 -6958.18,E2 -6958.18} C_VEL
LIN {X 0,Y 489.07,Z 222.428,A -85,B 0,C 180,E1 -6959.244,E2 -6959.244} C_VEL
LIN {X 0,Y 483.7,Z 204.437,A -85,B 0,C 180,E1 -6961.535,E2 -6961.535} C_VEL
LIN {X 0,Y 481.656,Z 197.786,A -85,B 0,C 180,E1 -6962.426,E2 -6962.426} C_VEL
LIN {X 0,Y 481.645,Z 197.802,A -85,B 0,C 180,E1 -6965.202,E2 -6965.202} C_VEL
LIN {X 0,Y 481.651,Z 197.803,A -85,B 0,C 180,E1 -6968.857,E2 -6968.857} C_VEL
LIN {X 0,Y 481.631,Z 197.8,A -85,B 0,C 180,E1 -6971.91,E2 -6971.91} C_VEL
LIN {X 0,Y 481.637,Z 197.801,A -85,B 0,C 180,E1 -6974.455,E2 -6974.455} C_VEL
LIN {X 0,Y 481.653,Z 197.799,A -85,B 0,C 180,E1 -6976.845,E2 -6976.845} C_VEL
LIN {X 0,Y 481.662,Z 197.795,A -85,B 0,C 180,E1 -6980.059,E2 -6980.059} C_VEL
LIN {X 0,Y 481.601,Z 197.802,A -85,B 0,C 180,E1 -6983.251,E2 -6983.251} C_VEL
LIN {X 0,Y 481.681,Z 197.794,A -85,B 0,C 180,E1 -6986.328,E2 -6986.328} C_VEL
LIN {X 0,Y 481.622,Z 197.804,A -85,B 0,C 180,E1 -6989.416,E2 -6989.416} C_VEL
LIN {X 0,Y 481.67,Z 197.794,A -85,B 0,C 180,E1 -6992.167,E2 -6992.167} C_VEL
LIN {X 0,Y 481.688,Z 197.792,A -85,B 0,C 180,E1 -6994.969,E2 -6994.969} C_VEL
LIN {X 0,Y 481.643,Z 197.798,A -85,B 0,C 180,E1 -6997.705,E2 -6997.705} C_VEL
LIN {X 0,Y 481.676,Z 197.784,A -85,B 0,C 180,E1 -7000.392,E2 -7000.392} C_VEL
LIN {X 0,Y 481.659,Z 197.802,A -85,B 0,C 180,E1 -7003.033,E2 -7003.033} C_VEL
LIN {X 0,Y 481.657,Z 197.792,A -85,B 0,C 180,E1 -7005.638,E2 -7005.638} C_VEL
LIN {X 0,Y 481.764,Z 197.766,A -85,B 0,C 180,E1 -7008.216,E2 -7008.216} C_VEL
LIN {X 0,Y 481.73,Z 197.787,A -85,B 0,C 180,E1 -7011.612,E2 -7011.612} C_VEL
LIN {X 0,Y 481.795,Z 197.777,A -85,B 0,C 180,E1 -7014.14,E2 -7014.14} C_VEL
LIN {X 0,Y 481.894,Z 197.757,A -85,B 0,C 180,E1 -7017.493,E2 -7017.493} C_VEL
LIN {X 0,Y 481.903,Z 197.765,A -85,B 0,C 180,E1 -7020,E2 -7020} C_VEL
LIN {X 0,Y 481.894,Z 197.772,A -85,B 0,C 180,E1 -7022.508,E2 -7022.508} C_VEL
LIN {X 0,Y 481.788,Z 197.774,A -85,B 0,C 180,E1 -7025.861,E2 -7025.861} C_VEL
LIN {X 0,Y 481.731,Z 197.792,A -85,B 0,C 180,E1 -7028.389,E2 -7028.389} C_VEL
LIN {X 0,Y 481.72,Z 197.777,A -85,B 0,C 180,E1 -7031.786,E2 -7031.786} C_VEL
LIN {X 0,Y 481.712,Z 197.789,A -85,B 0,C 180,E1 -7035.226,E2 -7035.226} C_VEL
LIN {X 0,Y 481.682,Z 197.787,A -85,B 0,C 180,E1 -7038.723,E2 -7038.723} C_VEL
LIN {X 0,Y 481.624,Z 197.799,A -85,B 0,C 180,E1 -7041.396,E2 -7041.396} C_VEL
LIN {X 0,Y 481.654,Z 197.799,A -85,B 0,C 180,E1 -7044.115,E2 -7044.115} C_VEL
LIN {X 0,Y 481.719,Z 197.785,A -85,B 0,C 180,E1 -7047.141,E2 -7047.141} C_VEL
LIN {X 0,Y 481.652,Z 197.798,A -85,B 0,C 180,E1 -7049.743,E2 -7049.743} C_VEL
LIN {X 0,Y 481.646,Z 197.792,A -85,B 0,C 180,E1 -7052.677,E2 -7052.677} C_VEL
LIN {X 0,Y 481.618,Z 197.802,A -85,B 0,C 180,E1 -7055.712,E2 -7055.712} C_VEL
LIN {X 0,Y 481.647,Z 197.789,A -85,B 0,C 180,E1 -7058.862,E2 -7058.862} C_VEL
LIN {X 0,Y 481.633,Z 197.802,A -85,B 0,C 180,E1 -7061.916,E2 -7061.916} C_VEL
LIN {X 0,Y 481.636,Z 197.795,A -85,B 0,C 180,E1 -7064.461,E2 -7064.461} C_VEL
LIN {X 0,Y 481.626,Z 197.804,A -85,B 0,C 180,E1 -7067.842,E2 -7067.842} C_VEL
LIN {X 0,Y 481.644,Z 197.796,A -85,B 0,C 180,E1 -7070.657,E2 -7070.657} C_VEL
LIN {X 0,Y 481.617,Z 197.802,A -85,B 0,C 180,E1 -7073.379,E2 -7073.379} C_VEL
LIN {X 0,Y 481.699,Z 197.794,A -85,B 0,C 180,E1 -7076.333,E2 -7076.333} C_VEL
LIN {X 0,Y 481.64,Z 197.798,A -85,B 0,C 180,E1 -7079.421,E2 -7079.421} C_VEL
LIN {X 0,Y 481.657,Z 197.803,A -85,B 0,C 180,E1 -7082.169,E2 -7082.169} C_VEL
LIN {X 0,Y 481.667,Z 197.794,A -85,B 0,C 180,E1 -7084.97,E2 -7084.97} C_VEL
LIN {X 0,Y 481.628,Z 197.8,A -85,B 0,C 180,E1 -7088.018,E2 -7088.018} C_VEL
LIN {X 0,Y 480.965,Z 197.886,A -85,B 0,C 180,E1 -7088.716,E2 -7088.716} C_VEL
LIN {X 0,Y 478.142,Z 198.241,A -85,B 0,C 180,E1 -7089.85,E2 -7089.85} C_VEL
LIN {X 0,Y 475.752,Z 198.533,A -85,B 0,C 180,E1 -7090.764,E2 -7090.764} C_VEL
LIN {X 0,Y 474.721,Z 198.661,A -85,B 0,C 180,E1 -7091.47,E2 -7091.47} C_VEL
LIN {X 0,Y 474.635,Z 198.675,A -85,B 0,C 180,E1 -7091.709,E2 -7091.709} C_VEL
LIN {X 0,Y 474.687,Z 198.668,A -85,B 0,C 180,E1 -7094.547,E2 -7094.547} C_VEL
LIN {X 0,Y 474.705,Z 198.666,A -85,B 0,C 180,E1 -7098.04,E2 -7098.04} C_VEL
LIN {X 0,Y 474.698,Z 198.669,A -85,B 0,C 180,E1 -7101.488,E2 -7101.488} C_VEL
LIN {X 0,Y 474.741,Z 198.654,A -85,B 0,C 180,E1 -7104.054,E2 -7104.054} C_VEL
LIN {X 0,Y 474.667,Z 198.706,A -85,B 0,C 180,E1 -7106.766,E2 -7106.766} C_VEL
LIN {X 0,Y 477.548,Z 208.423,A -85,B 0,C 180,E1 -7108.172,E2 -7108.172} C_VEL
LIN {X 0,Y 486.228,Z 227.273,A -85,B 0,C 180,E1 -7109.052,E2 -7109.052} C_VEL
LIN {X 0,Y 486.493,Z 230.502,A -85,B 0,C 180,E1 -7109.123,E2 -7109.123} C_VEL
LIN {X 0,Y 483.932,Z 413.996,A -85,B 0,C 180,E1 -7112.005,E2 -7112.005} C_VEL
LIN {X 0,Y 483.4,Z 430.452,A -85,B 0,C 180,E1 -7112.424,E2 -7112.424} C_VEL
LIN {X 0,Y 482.758,Z 445.891,A -85,B 0,C 180,E1 -7112.975,E2 -7112.975} C_VEL
LIN {X 0,Y 481.961,Z 460.827,A -85,B 0,C 180,E1 -7113.66,E2 -7113.66} C_VEL
LIN {X 0,Y 481.095,Z 475.488,A -85,B 0,C 180,E1 -7114.505,E2 -7114.505} C_VEL
LIN {X 0,Y 480.095,Z 489.346,A -85,B 0,C 180,E1 -7115.471,E2 -7115.471} C_VEL
LIN {X 0,Y 479.035,Z 503.368,A -85,B 0,C 180,E1 -7116.636,E2 -7116.636} C_VEL
LIN {X 0,Y 478.114,Z 515.438,A -85,B 0,C 180,E1 -7117.816,E2 -7117.816} C_VEL
LIN {X 0,Y 477.097,Z 528.464,A -85,B 0,C 180,E1 -7119.327,E2 -7119.327} C_VEL
LIN {X 0,Y 476.21,Z 539.547,A -85,B 0,C 180,E1 -7120.847,E2 -7120.847} C_VEL
LIN {X 0,Y 475.44,Z 549.856,A -85,B 0,C 180,E1 -7122.513,E2 -7122.513} C_VEL
LIN {X 0,Y 474.949,Z 558.365,A -85,B 0,C 180,E1 -7124.134,E2 -7124.134} C_VEL
LIN {X 0,Y 474.464,Z 566.414,A -85,B 0,C 180,E1 -7125.965,E2 -7125.965} C_VEL
LIN {X 0,Y 474.066,Z 574.055,A -85,B 0,C 180,E1 -7128.14,E2 -7128.14} C_VEL
LIN {X 0,Y 473.893,Z 578.945,A -85,B 0,C 180,E1 -7129.945,E2 -7129.945} C_VEL
LIN {X 0,Y 473.68,Z 582.74,A -85,B 0,C 180,E1 -7131.774,E2 -7131.774} C_VEL
LIN {X 0,Y 473.563,Z 585.441,A -85,B 0,C 180,E1 -7133.623,E2 -7133.623} C_VEL
LIN {X 0,Y 473.57,Z 586.927,A -85,B 0,C 180,E1 -7135.492,E2 -7135.492} C_VEL
LIN {X 0,Y 473.574,Z 587.312,A -85,B 0,C 180,E1 -7137.392,E2 -7137.392} C_VEL
LIN {X 0,Y 473.624,Z 586.531,A -85,B 0,C 180,E1 -7139.321,E2 -7139.321} C_VEL
LIN {X 0,Y 473.694,Z 584.404,A -85,B 0,C 180,E1 -7141.285,E2 -7141.285} C_VEL
LIN {X 0,Y 473.779,Z 580.909,A -85,B 0,C 180,E1 -7143.289,E2 -7143.289} C_VEL
LIN {X 0,Y 473.922,Z 577.347,A -85,B 0,C 180,E1 -7144.816,E2 -7144.816} C_VEL
LIN {X 0,Y 474.257,Z 571.183,A -85,B 0,C 180,E1 -7146.848,E2 -7146.848} C_VEL
LIN {X 0,Y 474.622,Z 563.991,A -85,B 0,C 180,E1 -7148.729,E2 -7148.729} C_VEL
LIN {X 0,Y 475.116,Z 555.221,A -85,B 0,C 180,E1 -7150.607,E2 -7150.607} C_VEL
LIN {X 0,Y 475.81,Z 545.167,A -85,B 0,C 180,E1 -7152.393,E2 -7152.393} C_VEL
LIN {X 0,Y 476.701,Z 534.339,A -85,B 0,C 180,E1 -7154.009,E2 -7154.009} C_VEL
LIN {X 0,Y 477.63,Z 522.314,A -85,B 0,C 180,E1 -7155.532,E2 -7155.532} C_VEL
LIN {X 0,Y 478.686,Z 508.937,A -85,B 0,C 180,E1 -7156.957,E2 -7156.957} C_VEL
LIN {X 0,Y 479.766,Z 494.741,A -85,B 0,C 180,E1 -7158.22,E2 -7158.22} C_VEL
LIN {X 0,Y 480.768,Z 480.629,A -85,B 0,C 180,E1 -7159.269,E2 -7159.269} C_VEL
LIN {X 0,Y 481.745,Z 466.332,A -85,B 0,C 180,E1 -7160.15,E2 -7160.15} C_VEL
LIN {X 0,Y 482.567,Z 451.885,A -85,B 0,C 180,E1 -7160.881,E2 -7160.881} C_VEL
LIN {X 0,Y 483.273,Z 436.353,A -85,B 0,C 180,E1 -7161.491,E2 -7161.491} C_VEL
LIN {X 0,Y 483.835,Z 419.711,A -85,B 0,C 180,E1 -7161.972,E2 -7161.972} C_VEL
LIN {X 0,Y 484.225,Z 399.779,A -85,B 0,C 180,E1 -7162.343,E2 -7162.343} C_VEL
LIN {X 0,Y 486.608,Z 228.513,A -85,B 0,C 180,E1 -7165.034,E2 -7165.034} C_VEL
LIN {X 0,Y 484.607,Z 223.457,A -85,B 0,C 180,E1 -7165.249,E2 -7165.249} C_VEL
LIN {X 0,Y 477.747,Z 209.016,A -85,B 0,C 180,E1 -7165.961,E2 -7165.961} C_VEL
LIN {X 0,Y 474.643,Z 198.676,A -85,B 0,C 180,E1 -7167.502,E2 -7167.502} C_VEL
LIN {X 0,Y 474.626,Z 198.676,A -85,B 0,C 180,E1 -7170.884,E2 -7170.884} C_VEL
LIN {X 0,Y 474.656,Z 198.671,A -85,B 0,C 180,E1 -7173.628,E2 -7173.628} C_VEL
LIN {X 0,Y 474.636,Z 198.675,A -85,B 0,C 180,E1 -7176.641,E2 -7176.641} C_VEL
LIN {X 0,Y 474.656,Z 198.673,A -85,B 0,C 180,E1 -7180.089,E2 -7180.089} C_VEL
LIN {X 0,Y 474.65,Z 198.667,A -85,B 0,C 180,E1 -7182.774,E2 -7182.774} C_VEL
LIN {X 0,Y 474.647,Z 198.672,A -85,B 0,C 180,E1 -7185.42,E2 -7185.42} C_VEL
LIN {X 0,Y 474.704,Z 198.67,A -85,B 0,C 180,E1 -7188.037,E2 -7188.037} C_VEL
LIN {X 0,Y 474.725,Z 198.664,A -85,B 0,C 180,E1 -7191.486,E2 -7191.486} C_VEL
LIN {X 0,Y 474.776,Z 198.658,A -85,B 0,C 180,E1 -7194.052,E2 -7194.052} C_VEL
LIN {X 0,Y 474.89,Z 198.643,A -85,B 0,C 180,E1 -7197.455,E2 -7197.455} C_VEL
LIN {X 0,Y 474.908,Z 198.642,A -85,B 0,C 180,E1 -7200,E2 -7200} C_VEL
LIN {X 0,Y 474.89,Z 198.64,A -85,B 0,C 180,E1 -7202.544,E2 -7202.544} C_VEL
LIN {X 0,Y 474.766,Z 198.659,A -85,B 0,C 180,E1 -7205.947,E2 -7205.947} C_VEL
LIN {X 0,Y 474.71,Z 198.662,A -85,B 0,C 180,E1 -7208.513,E2 -7208.513} C_VEL
LIN {X 0,Y 474.702,Z 198.665,A -85,B 0,C 180,E1 -7211.962,E2 -7211.962} C_VEL
LIN {X 0,Y 474.698,Z 198.668,A -85,B 0,C 180,E1 -7215.455,E2 -7215.455} C_VEL
LIN {X 0,Y 474.661,Z 198.67,A -85,B 0,C 180,E1 -7219.01,E2 -7219.01} C_VEL
LIN {X 0,Y 474.586,Z 198.68,A -85,B 0,C 180,E1 -7221.729,E2 -7221.729} C_VEL
LIN {X 0,Y 474.637,Z 198.669,A -85,B 0,C 180,E1 -7224.494,E2 -7224.494} C_VEL
LIN {X 0,Y 474.679,Z 198.67,A -85,B 0,C 180,E1 -7227.334,E2 -7227.334} C_VEL
LIN {X 0,Y 474.602,Z 198.679,A -85,B 0,C 180,E1 -7230.809,E2 -7230.809} C_VEL
LIN {X 0,Y 474.62,Z 198.672,A -85,B 0,C 180,E1 -7233.98,E2 -7233.98} C_VEL
LIN {X 0,Y 474.571,Z 198.683,A -85,B 0,C 180,E1 -7236.899,E2 -7236.899} C_VEL
LIN {X 0,Y 474.607,Z 198.677,A -85,B 0,C 180,E1 -7239.644,E2 -7239.644} C_VEL
LIN {X 0,Y 474.6,Z 198.676,A -85,B 0,C 180,E1 -7242.233,E2 -7242.233} C_VEL
LIN {X 0,Y 474.616,Z 198.678,A -85,B 0,C 180,E1 -7245.297,E2 -7245.297} C_VEL
LIN {X 0,Y 474.604,Z 198.676,A -85,B 0,C 180,E1 -7248.212,E2 -7248.212} C_VEL
LIN {X 0,Y 474.609,Z 198.678,A -85,B 0,C 180,E1 -7251.542,E2 -7251.542} C_VEL
LIN {X 0,Y 474.623,Z 198.676,A -85,B 0,C 180,E1 -7254.725,E2 -7254.725} C_VEL
LIN {X 0,Y 474.65,Z 198.758,A -85,B 0,C 180,E1 -7257.154,E2 -7257.154} C_VEL
LIN {X 0,Y 480.174,Z 216.528,A -85,B 0,C 180,E1 -7259.551,E2 -7259.551} C_VEL
LIN {X 0,Y 482.269,Z 224.022,A -85,B 0,C 180,E1 -7260.51,E2 -7260.51} C_VEL
LIN {X 0,Y 482.34,Z 228.075,A -85,B 0,C 180,E1 -7260.954,E2 -7260.954} C_VEL
LIN {X 0,Y 482.071,Z 232.035,A -85,B 0,C 180,E1 -7261.365,E2 -7261.365} C_VEL
LIN {X 0,Y 486.309,Z 256.202,A -85,B 0,C 180,E1 -7262.05,E2 -7262.05} C_VEL
LIN {X 0,Y 484.959,Z 351.184,A -85,B 0,C 180,E1 -7263.543,E2 -7263.543} C_VEL
LIN {X 0,Y 483.797,Z 438.71,A -85,B 0,C 180,E1 -7264.928,E2 -7264.928} C_VEL
LIN {X 0,Y 483.176,Z 455.218,A -85,B 0,C 180,E1 -7265.336,E2 -7265.336} C_VEL
LIN {X 0,Y 482.451,Z 471.865,A -85,B 0,C 180,E1 -7265.927,E2 -7265.927} C_VEL
LIN {X 0,Y 481.638,Z 486.007,A -85,B 0,C 180,E1 -7266.569,E2 -7266.569} C_VEL
LIN {X 0,Y 480.679,Z 501.145,A -85,B 0,C 180,E1 -7267.433,E2 -7267.433} C_VEL
LIN {X 0,Y 479.656,Z 515.101,A -85,B 0,C 180,E1 -7268.398,E2 -7268.398} C_VEL
LIN {X 0,Y 478.544,Z 529.726,A -85,B 0,C 180,E1 -7269.607,E2 -7269.607} C_VEL
LIN {X 0,Y 477.497,Z 542.801,A -85,B 0,C 180,E1 -7270.889,E2 -7270.889} C_VEL
LIN {X 0,Y 476.67,Z 554.052,A -85,B 0,C 180,E1 -7272.184,E2 -7272.184} C_VEL
LIN {X 0,Y 475.856,Z 565.595,A -85,B 0,C 180,E1 -7273.738,E2 -7273.738} C_VEL
LIN {X 0,Y 475.124,Z 576.293,A -85,B 0,C 180,E1 -7275.434,E2 -7275.434} C_VEL
LIN {X 0,Y 474.635,Z 585.496,A -85,B 0,C 180,E1 -7277.166,E2 -7277.166} C_VEL
LIN {X 0,Y 474.245,Z 593.197,A -85,B 0,C 180,E1 -7278.891,E2 -7278.891} C_VEL
LIN {X 0,Y 473.945,Z 600.932,A -85,B 0,C 180,E1 -7281.041,E2 -7281.041} C_VEL
LIN {X 0,Y 473.823,Z 606.818,A -85,B 0,C 180,E1 -7283.183,E2 -7283.183} C_VEL
LIN {X 0,Y 473.759,Z 610.262,A -85,B 0,C 180,E1 -7284.892,E2 -7284.892} C_VEL
LIN {X 0,Y 473.74,Z 612.767,A -85,B 0,C 180,E1 -7286.596,E2 -7286.596} C_VEL
LIN {X 0,Y 473.719,Z 614.183,A -85,B 0,C 180,E1 -7288.298,E2 -7288.298} C_VEL
LIN {X 0,Y 473.664,Z 614.719,A -85,B 0,C 180,E1 -7289.998,E2 -7289.998} C_VEL
LIN {X 0,Y 473.718,Z 614.197,A -85,B 0,C 180,E1 -7291.698,E2 -7291.698} C_VEL
LIN {X 0,Y 473.738,Z 612.795,A -85,B 0,C 180,E1 -7293.4,E2 -7293.4} C_VEL
LIN {X 0,Y 473.758,Z 610.307,A -85,B 0,C 180,E1 -7295.104,E2 -7295.104} C_VEL
LIN {X 0,Y 473.819,Z 606.882,A -85,B 0,C 180,E1 -7296.813,E2 -7296.813} C_VEL
LIN {X 0,Y 473.951,Z 601.02,A -85,B 0,C 180,E1 -7298.955,E2 -7298.955} C_VEL
LIN {X 0,Y 474.254,Z 593.307,A -85,B 0,C 180,E1 -7301.105,E2 -7301.105} C_VEL
LIN {X 0,Y 474.672,Z 584.605,A -85,B 0,C 180,E1 -7303.047,E2 -7303.047} C_VEL
LIN {X 0,Y 475.249,Z 575.208,A -85,B 0,C 180,E1 -7304.776,E2 -7304.776} C_VEL
LIN {X 0,Y 475.892,Z 565.532,A -85,B 0,C 180,E1 -7306.293,E2 -7306.293} C_VEL
LIN {X 0,Y 476.677,Z 554.253,A -85,B 0,C 180,E1 -7307.811,E2 -7307.811} C_VEL
LIN {X 0,Y 477.627,Z 542.033,A -85,B 0,C 180,E1 -7309.213,E2 -7309.213} C_VEL
LIN {X 0,Y 478.628,Z 528.661,A -85,B 0,C 180,E1 -7310.508,E2 -7310.508} C_VEL
LIN {X 0,Y 479.625,Z 515.341,A -85,B 0,C 180,E1 -7311.599,E2 -7311.599} C_VEL
LIN {X 0,Y 480.788,Z 500.127,A -85,B 0,C 180,E1 -7312.638,E2 -7312.638} C_VEL
LIN {X 0,Y 481.713,Z 485.17,A -85,B 0,C 180,E1 -7313.48,E2 -7313.48} C_VEL
LIN {X 0,Y 482.645,Z 468.161,A -85,B 0,C 180,E1 -7314.23,E2 -7314.23} C_VEL
LIN {X 0,Y 483.335,Z 451.723,A -85,B 0,C 180,E1 -7314.765,E2 -7314.765} C_VEL
LIN {X 0,Y 483.875,Z 435.866,A -85,B 0,C 180,E1 -7315.118,E2 -7315.118} C_VEL
LIN {X 0,Y 486.332,Z 257.201,A -85,B 0,C 180,E1 -7317.912,E2 -7317.912} C_VEL
LIN {X 0,Y 482.634,Z 235.987,A -85,B 0,C 180,E1 -7318.495,E2 -7318.495} C_VEL
LIN {X 0,Y 482.064,Z 232.311,A -85,B 0,C 180,E1 -7318.62,E2 -7318.62} C_VEL
LIN {X 0,Y 482.507,Z 226.022,A -85,B 0,C 180,E1 -7319.267,E2 -7319.267} C_VEL
LIN {X 0,Y 482.339,Z 224.094,A -85,B 0,C 180,E1 -7319.485,E2 -7319.485} C_VEL
LIN {X 0,Y 477.04,Z 206.556,A -85,B 0,C 180,E1 -7321.761,E2 -7321.761} C_VEL
LIN {X 0,Y 474.607,Z 198.663,A -85,B 0,C 180,E1 -7322.841,E2 -7322.841} C_VEL
LIN {X 0,Y 474.597,Z 198.679,A -85,B 0,C 180,E1 -7325.467,E2 -7325.467} C_VEL
LIN {X 0,Y 474.592,Z 198.68,A -85,B 0,C 180,E1 -7328.455,E2 -7328.455} C_VEL
LIN {X 0,Y 474.599,Z 198.677,A -85,B 0,C 180,E1 -7331.783,E2 -7331.783} C_VEL
LIN {X 0,Y 474.598,Z 198.68,A -85,B 0,C 180,E1 -7334.701,E2 -7334.701} C_VEL
LIN {X 0,Y 474.608,Z 198.677,A -85,B 0,C 180,E1 -7337.76,E2 -7337.76} C_VEL
LIN {X 0,Y 474.64,Z 198.67,A -85,B 0,C 180,E1 -7340.454,E2 -7340.454} C_VEL
LIN {X 0,Y 474.565,Z 198.677,A -85,B 0,C 180,E1 -7343.675,E2 -7343.675} C_VEL
LIN {X 0,Y 474.615,Z 198.678,A -85,B 0,C 180,E1 -7346.778,E2 -7346.778} C_VEL
LIN {X 0,Y 474.576,Z 198.679,A -85,B 0,C 180,E1 -7349.768,E2 -7349.768} C_VEL
LIN {X 0,Y 474.667,Z 198.668,A -85,B 0,C 180,E1 -7352.678,E2 -7352.678} C_VEL
LIN {X 0,Y 474.631,Z 198.673,A -85,B 0,C 180,E1 -7355.506,E2 -7355.506} C_VEL
LIN {X 0,Y 474.644,Z 198.663,A -85,B 0,C 180,E1 -7359.185,E2 -7359.185} C_VEL
LIN {X 0,Y 474.624,Z 198.668,A -85,B 0,C 180,E1 -7361.883,E2 -7361.883} C_VEL
LIN {X 0,Y 474.666,Z 198.672,A -85,B 0,C 180,E1 -7364.544,E2 -7364.544} C_VEL
LIN {X 0,Y 474.707,Z 198.643,A -85,B 0,C 180,E1 -7368.038,E2 -7368.038} C_VEL
LIN {X 0,Y 474.696,Z 198.664,A -85,B 0,C 180,E1 -7371.486,E2 -7371.486} C_VEL
